KUKA KRL program: EPS_2_251524_MH1A_A_20251121061154.src

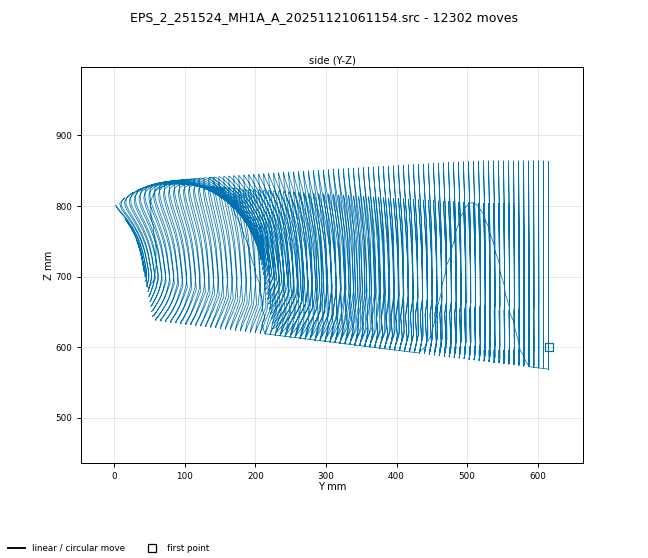
[picture p0: tool path of EPS_2_251524_MH1A_A_20251121061154.src, 12302 of 12304 moves have a stored position in this frame; points joined in program order, loops and branches not executed]
&ACCESS RVP
&REL 4
&COMMENT QRS 19112012
&PARAM EDITMASK = *
DEF PART()
EXT BAS (BAS_COMMAND :IN,REAL :IN )
INT I
BAS (#INITMOV,0 )

;KUKA QRS Post kuka4.cps  Date:22-06-2017 !

File_ID=2928

QRS_PRE_INIT()

;Init var - Until changes are made in qrs_pre_init
Outlet_Square_prg=0
Inlet_1_Square_prg=0
Inlet_2_Square_prg=0
Inlet_3_Square_prg=0
Inlet_4_Square_prg=0
Inlet_5_Square_prg=0

Outlet_1={X 0.000, Y 513.730, Z 763.500, B 0.000, E1 0.000 }
Inlet_1={X 0.000, Y 518.010, Z 703.500, B 0.000, E1 125.000 }
Outlet_1_type=201
Inlet_1_type=201
;QRS#1=Sidecore dimensions
;QRS#2=200-8" PVC SDR 35
;QRS#3=200-8" PVC SDR 35
;QRS#4=
;QRS#5=
;QRS#6=
;QRS#7=
;QRS#8=
;QRS#9=12-08 PSX
;QRS#10=12-08 PSX
;QRS#11=
;QRS#12=
;QRS#13=
;QRS#14=
;QRS#15=
;QRS#16=1220x127x1143 3,75'
;QRS#17=EPS Height
;QRS#18=864
;QRS#19=*
;QRS#20= UPDATED VERSION 22-06-2017
;QRS#21=*
Outlet_Square=0100
Inlet_1_Square=0100
Inlet_2_Square=0
Inlet_3_Square=0
Inlet_4_Square=0
Inlet_5_Square=0
Mill_Square=1
Outlet_Square_Prg=204
Inlet_1_Square_prg=204

QRS_INIT()

$ADVANCE=5

; T1
PTP {E1 173.595,E2 173.595}
PTP {X 0,Y 615.511,A -85,B 0,C 180,E1 173.595,E2 173.595,E3 0,E4 0,E5 0,E6 0}
QRS_SPEED_INIT()
LIN {X 0,Y 615.511,Z 600,A -85,B 0,C 180,E1 173.595,E2 173.595,E3 0,E4 0,E5 0,E6 0} C_VEL
LIN {X 0,Y 615.511,Z 578.873,A -85,B 0,C 180,E1 173.595,E2 173.595} C_VEL
LIN {X 0,Y 615.511,Z 570.691,A -85,B 0,C 180,E1 173.595,E2 173.595} C_VEL
LIN {X 0,Y 615.492,Z 568.691,A -85,B 0,C 180,E1 173.409,E2 173.409} C_VEL
LIN {X 0,Y 615.475,Z 568.685,A -85,B 0,C 180,E1 170.801,E2 170.801} C_VEL
LIN {X 0,Y 615.486,Z 568.69,A -85,B 0,C 180,E1 168.139,E2 168.139} C_VEL
LIN {X 0,Y 615.493,Z 568.691,A -85,B 0,C 180,E1 165.451,E2 165.451} C_VEL
LIN {X 0,Y 615.476,Z 568.685,A -85,B 0,C 180,E1 162.729,E2 162.729} C_VEL
LIN {X 0,Y 615.485,Z 568.748,A -85,B 0,C 180,E1 162.301,E2 162.301} C_VEL
LIN {X 0,Y 615.48,Z 584.538,A -85,B 0,C 180,E1 159.442,E2 159.442} C_VEL
LIN {X 0,Y 615.48,Z 593.631,A -85,B 0,C 180,E1 157.811,E2 157.811} C_VEL
LIN {X 0,Y 615.477,Z 700.494,A -85,B 0,C 180,E1 156.532,E2 156.532} C_VEL
LIN {X 0,Y 615.486,Z 713.363,A -85,B 0,C 180,E1 156.245,E2 156.245} C_VEL
LIN {X 0,Y 615.488,Z 725.164,A -85,B 0,C 180,E1 155.859,E2 155.859} C_VEL
LIN {X 0,Y 615.492,Z 736.391,A -85,B 0,C 180,E1 155.369,E2 155.369} C_VEL
LIN {X 0,Y 615.486,Z 747.967,A -85,B 0,C 180,E1 154.718,E2 154.718} C_VEL
LIN {X 0,Y 615.499,Z 759.136,A -85,B 0,C 180,E1 153.921,E2 153.921} C_VEL
LIN {X 0,Y 615.499,Z 768.418,A -85,B 0,C 180,E1 153.103,E2 153.103} C_VEL
LIN {X 0,Y 615.493,Z 777.665,A -85,B 0,C 180,E1 152.085,E2 152.085} C_VEL
LIN {X 0,Y 615.498,Z 784.494,A -85,B 0,C 180,E1 151.156,E2 151.156} C_VEL
LIN {X 0,Y 615.499,Z 790.175,A -85,B 0,C 180,E1 150.202,E2 150.202} C_VEL
LIN {X 0,Y 615.497,Z 795.401,A -85,B 0,C 180,E1 149.081,E2 149.081} C_VEL
LIN {X 0,Y 615.495,Z 798.12,A -85,B 0,C 180,E1 148.315,E2 148.315} C_VEL
LIN {X 0,Y 615.493,Z 800.307,A -85,B 0,C 180,E1 147.543,E2 147.543} C_VEL
LIN {X 0,Y 615.495,Z 802.346,A -85,B 0,C 180,E1 146.463,E2 146.463} C_VEL
LIN {X 0,Y 615.492,Z 803.34,A -85,B 0,C 180,E1 145.185,E2 145.185} C_VEL
LIN {X 0,Y 615.496,Z 803.076,A -85,B 0,C 180,E1 144.163,E2 144.163} C_VEL
LIN {X 0,Y 615.493,Z 801.724,A -85,B 0,C 180,E1 143.061,E2 143.061} C_VEL
LIN {X 0,Y 615.495,Z 799.15,A -85,B 0,C 180,E1 141.932,E2 141.932} C_VEL
LIN {X 0,Y 615.496,Z 795.8,A -85,B 0,C 180,E1 140.935,E2 140.935} C_VEL
LIN {X 0,Y 615.496,Z 791.221,A -85,B 0,C 180,E1 139.909,E2 139.909} C_VEL
LIN {X 0,Y 615.495,Z 785.487,A -85,B 0,C 180,E1 138.903,E2 138.903} C_VEL
LIN {X 0,Y 615.494,Z 778.427,A -85,B 0,C 180,E1 137.918,E2 137.918} C_VEL
LIN {X 0,Y 615.495,Z 769.828,A -85,B 0,C 180,E1 136.95,E2 136.95} C_VEL
LIN {X 0,Y 615.495,Z 760.482,A -85,B 0,C 180,E1 136.095,E2 136.095} C_VEL
LIN {X 0,Y 615.49,Z 750.585,A -85,B 0,C 180,E1 135.363,E2 135.363} C_VEL
LIN {X 0,Y 615.489,Z 740.106,A -85,B 0,C 180,E1 134.734,E2 134.734} C_VEL
LIN {X 0,Y 615.49,Z 727.652,A -85,B 0,C 180,E1 134.148,E2 134.148} C_VEL
LIN {X 0,Y 615.496,Z 715.095,A -85,B 0,C 180,E1 133.713,E2 133.713} C_VEL
LIN {X 0,Y 615.479,Z 702.164,A -85,B 0,C 180,E1 133.408,E2 133.408} C_VEL
LIN {X 0,Y 615.477,Z 680.151,A -85,B 0,C 180,E1 133.121,E2 133.121} C_VEL
LIN {X 0,Y 615.477,Z 593.615,A -85,B 0,C 180,E1 132.096,E2 132.096} C_VEL
LIN {X 0,Y 615.482,Z 578.635,A -85,B 0,C 180,E1 129.404,E2 129.404} C_VEL
LIN {X 0,Y 615.49,Z 568.685,A -85,B 0,C 180,E1 127.577,E2 127.577} C_VEL
LIN {X 0,Y 615.49,Z 568.684,A -85,B 0,C 180,E1 124.701,E2 124.701} C_VEL
LIN {X 0,Y 615.492,Z 568.691,A -85,B 0,C 180,E1 122.331,E2 122.331} C_VEL
LIN {X 0,Y 615.492,Z 568.684,A -85,B 0,C 180,E1 119.405,E2 119.405} C_VEL
LIN {X 0,Y 615.474,Z 568.684,A -85,B 0,C 180,E1 117.043,E2 117.043} C_VEL
LIN {X 0,Y 615.495,Z 568.688,A -85,B 0,C 180,E1 114.271,E2 114.271} C_VEL
LIN {X 0,Y 615.492,Z 568.688,A -85,B 0,C 180,E1 111.431,E2 111.431} C_VEL
LIN {X 0,Y 615.478,Z 568.684,A -85,B 0,C 180,E1 108.602,E2 108.602} C_VEL
LIN {X 0,Y 615.492,Z 568.696,A -85,B 0,C 180,E1 105.904,E2 105.904} C_VEL
LIN {X 0,Y 615.497,Z 568.684,A -85,B 0,C 180,E1 103.2,E2 103.2} C_VEL
LIN {X 0,Y 615.476,Z 568.684,A -85,B 0,C 180,E1 100.526,E2 100.526} C_VEL
LIN {X 0,Y 615.493,Z 568.691,A -85,B 0,C 180,E1 97.875,E2 97.875} C_VEL
LIN {X 0,Y 615.486,Z 568.692,A -85,B 0,C 180,E1 95.24,E2 95.24} C_VEL
LIN {X 0,Y 615.477,Z 568.684,A -85,B 0,C 180,E1 92.617,E2 92.617} C_VEL
LIN {X 0,Y 615.489,Z 568.685,A -85,B 0,C 180,E1 89.999,E2 89.999} C_VEL
LIN {X 0,Y 615.495,Z 568.7,A -85,B 0,C 180,E1 87.381,E2 87.381} C_VEL
LIN {X 0,Y 615.485,Z 568.685,A -85,B 0,C 180,E1 84.758,E2 84.758} C_VEL
LIN {X 0,Y 615.481,Z 568.683,A -85,B 0,C 180,E1 82.124,E2 82.124} C_VEL
LIN {X 0,Y 615.49,Z 568.694,A -85,B 0,C 180,E1 79.472,E2 79.472} C_VEL
LIN {X 0,Y 615.497,Z 568.686,A -85,B 0,C 180,E1 76.798,E2 76.798} C_VEL
LIN {X 0,Y 615.478,Z 568.683,A -85,B 0,C 180,E1 74.094,E2 74.094} C_VEL
LIN {X 0,Y 615.491,Z 568.693,A -85,B 0,C 180,E1 71.353,E2 71.353} C_VEL
LIN {X 0,Y 615.492,Z 568.686,A -85,B 0,C 180,E1 68.568,E2 68.568} C_VEL
LIN {X 0,Y 615.489,Z 568.682,A -85,B 0,C 180,E1 65.727,E2 65.727} C_VEL
LIN {X 0,Y 615.494,Z 568.696,A -85,B 0,C 180,E1 62.823,E2 62.823} C_VEL
LIN {X 0,Y 615.476,Z 568.685,A -85,B 0,C 180,E1 60.207,E2 60.207} C_VEL
LIN {X 0,Y 615.486,Z 568.684,A -85,B 0,C 180,E1 57.542,E2 57.542} C_VEL
LIN {X 0,Y 615.492,Z 568.689,A -85,B 0,C 180,E1 55.185,E2 55.185} C_VEL
LIN {X 0,Y 615.491,Z 568.701,A -85,B 0,C 180,E1 52.758,E2 52.758} C_VEL
LIN {X 0,Y 615.477,Z 568.684,A -85,B 0,C 180,E1 49.912,E2 49.912} C_VEL
LIN {X 0,Y 615.478,Z 568.683,A -85,B 0,C 180,E1 47.646,E2 47.646} C_VEL
LIN {X 0,Y 615.49,Z 568.691,A -85,B 0,C 180,E1 44.931,E2 44.931} C_VEL
LIN {X 0,Y 615.49,Z 568.686,A -85,B 0,C 180,E1 42.08,E2 42.08} C_VEL
LIN {X 0,Y 615.474,Z 568.685,A -85,B 0,C 180,E1 39.751,E2 39.751} C_VEL
LIN {X 0,Y 615.489,Z 568.687,A -85,B 0,C 180,E1 36.936,E2 36.936} C_VEL
LIN {X 0,Y 615.495,Z 568.687,A -85,B 0,C 180,E1 34.021,E2 34.021} C_VEL
LIN {X 0,Y 615.478,Z 568.685,A -85,B 0,C 180,E1 31.686,E2 31.686} C_VEL
LIN {X 0,Y 615.477,Z 568.683,A -85,B 0,C 180,E1 29.407,E2 29.407} C_VEL
LIN {X 0,Y 615.488,Z 568.682,A -85,B 0,C 180,E1 27.044,E2 27.044} C_VEL
LIN {X 0,Y 615.488,Z 568.702,A -85,B 0,C 180,E1 24.272,E2 24.272} C_VEL
LIN {X 0,Y 615.477,Z 568.685,A -85,B 0,C 180,E1 21.432,E2 21.432} C_VEL
LIN {X 0,Y 615.486,Z 568.687,A -85,B 0,C 180,E1 18.646,E2 18.646} C_VEL
LIN {X 0,Y 615.489,Z 568.695,A -85,B 0,C 180,E1 15.905,E2 15.905} C_VEL
LIN {X 0,Y 615.476,Z 568.684,A -85,B 0,C 180,E1 13.201,E2 13.201} C_VEL
LIN {X 0,Y 615.489,Z 568.685,A -85,B 0,C 180,E1 10.527,E2 10.527} C_VEL
LIN {X 0,Y 615.493,Z 568.698,A -85,B 0,C 180,E1 7.875,E2 7.875} C_VEL
LIN {X 0,Y 615.478,Z 568.686,A -85,B 0,C 180,E1 5.241,E2 5.241} C_VEL
LIN {X 0,Y 615.494,Z 568.681,A -85,B 0,C 180,E1 2.618,E2 2.618} C_VEL
LIN {X 0,Y 615.491,Z 568.695,A -85,B 0,C 180,E1 0,E2 0} C_VEL
LIN {X 0,Y 615.494,Z 568.688,A -85,B 0,C 180,E1 -2.618,E2 -2.618} C_VEL
LIN {X 0,Y 615.477,Z 568.683,A -85,B 0,C 180,E1 -5.241,E2 -5.241} C_VEL
LIN {X 0,Y 615.489,Z 568.687,A -85,B 0,C 180,E1 -7.876,E2 -7.876} C_VEL
LIN {X 0,Y 615.484,Z 568.687,A -85,B 0,C 180,E1 -10.885,E2 -10.885} C_VEL
LIN {X 0,Y 615.476,Z 568.685,A -85,B 0,C 180,E1 -13.202,E2 -13.202} C_VEL
LIN {X 0,Y 615.487,Z 568.685,A -85,B 0,C 180,E1 -15.905,E2 -15.905} C_VEL
LIN {X 0,Y 615.494,Z 568.697,A -85,B 0,C 180,E1 -18.646,E2 -18.646} C_VEL
LIN {X 0,Y 615.476,Z 568.684,A -85,B 0,C 180,E1 -21.432,E2 -21.432} C_VEL
LIN {X 0,Y 615.487,Z 568.69,A -85,B 0,C 180,E1 -24.272,E2 -24.272} C_VEL
LIN {X 0,Y 615.48,Z 568.688,A -85,B 0,C 180,E1 -27.178,E2 -27.178} C_VEL
LIN {X 0,Y 615.485,Z 568.682,A -85,B 0,C 180,E1 -29.793,E2 -29.793} C_VEL
LIN {X 0,Y 615.487,Z 568.691,A -85,B 0,C 180,E1 -32.458,E2 -32.458} C_VEL
LIN {X 0,Y 615.498,Z 568.7,A -85,B 0,C 180,E1 -34.815,E2 -34.815} C_VEL
LIN {X 0,Y 615.49,Z 568.689,A -85,B 0,C 180,E1 -37.242,E2 -37.242} C_VEL
LIN {X 0,Y 615.493,Z 568.68,A -85,B 0,C 180,E1 -40.089,E2 -40.089} C_VEL
LIN {X 0,Y 615.496,Z 568.698,A -85,B 0,C 180,E1 -43.048,E2 -43.048} C_VEL
LIN {X 0,Y 615.481,Z 568.682,A -85,B 0,C 180,E1 -46.003,E2 -46.003} C_VEL
LIN {X 0,Y 615.489,Z 568.696,A -85,B 0,C 180,E1 -48.906,E2 -48.906} C_VEL
LIN {X 0,Y 615.495,Z 568.7,A -85,B 0,C 180,E1 -51.096,E2 -51.096} C_VEL
LIN {X 0,Y 615.482,Z 568.69,A -85,B 0,C 180,E1 -53.574,E2 -53.574} C_VEL
LIN {X 0,Y 615.475,Z 568.685,A -85,B 0,C 180,E1 -55.977,E2 -55.977} C_VEL
LIN {X 0,Y 615.487,Z 568.681,A -85,B 0,C 180,E1 -58.314,E2 -58.314} C_VEL
LIN {X 0,Y 615.494,Z 568.681,A -85,B 0,C 180,E1 -60.593,E2 -60.593} C_VEL
LIN {X 0,Y 615.494,Z 568.693,A -85,B 0,C 180,E1 -63.556,E2 -63.556} C_VEL
LIN {X 0,Y 615.487,Z 568.681,A -85,B 0,C 180,E1 -66.443,E2 -66.443} C_VEL
LIN {X 0,Y 615.492,Z 568.868,A -85,B 0,C 180,E1 -66.711,E2 -66.711} C_VEL
LIN {X 0,Y 615.487,Z 591.047,A -85,B 0,C 180,E1 -69.575,E2 -69.575} C_VEL
LIN {X 0,Y 615.484,Z 613.193,A -85,B 0,C 180,E1 -72.386,E2 -72.386} C_VEL
LIN {X 0,Y 615.481,Z 634.978,A -85,B 0,C 180,E1 -75.112,E2 -75.112} C_VEL
LIN {X 0,Y 615.478,Z 651.127,A -85,B 0,C 180,E1 -77.113,E2 -77.113} C_VEL
LIN {X 0,Y 615.476,Z 759.796,A -85,B 0,C 180,E1 -78.41,E2 -78.41} C_VEL
LIN {X 0,Y 615.487,Z 772.32,A -85,B 0,C 180,E1 -78.681,E2 -78.681} C_VEL
LIN {X 0,Y 615.496,Z 785.511,A -85,B 0,C 180,E1 -79.109,E2 -79.109} C_VEL
LIN {X 0,Y 615.484,Z 797.465,A -85,B 0,C 180,E1 -79.639,E2 -79.639} C_VEL
LIN {X 0,Y 615.483,Z 808.986,A -85,B 0,C 180,E1 -80.303,E2 -80.303} C_VEL
LIN {X 0,Y 615.499,Z 819.333,A -85,B 0,C 180,E1 -81.049,E2 -81.049} C_VEL
LIN {X 0,Y 615.497,Z 827.805,A -85,B 0,C 180,E1 -81.793,E2 -81.793} C_VEL
LIN {X 0,Y 615.498,Z 835.6,A -85,B 0,C 180,E1 -82.619,E2 -82.619} C_VEL
LIN {X 0,Y 615.496,Z 843.198,A -85,B 0,C 180,E1 -83.607,E2 -83.607} C_VEL
LIN {X 0,Y 615.498,Z 850.201,A -85,B 0,C 180,E1 -84.758,E2 -84.758} C_VEL
LIN {X 0,Y 615.494,Z 854.848,A -85,B 0,C 180,E1 -85.743,E2 -85.743} C_VEL
LIN {X 0,Y 615.496,Z 858.396,A -85,B 0,C 180,E1 -86.726,E2 -86.726} C_VEL
LIN {X 0,Y 615.497,Z 860.231,A -85,B 0,C 180,E1 -87.381,E2 -87.381} C_VEL
LIN {X 0,Y 615.496,Z 861.607,A -85,B 0,C 180,E1 -88.036,E2 -88.036} C_VEL
LIN {X 0,Y 615.496,Z 863.173,A -85,B 0,C 180,E1 -89.345,E2 -89.345} C_VEL
LIN {X 0,Y 615.494,Z 863.389,A -85,B 0,C 180,E1 -89.999,E2 -89.999} C_VEL
LIN {X 0,Y 615.496,Z 862.581,A -85,B 0,C 180,E1 -91.308,E2 -91.308} C_VEL
LIN {X 0,Y 615.496,Z 861.609,A -85,B 0,C 180,E1 -91.962,E2 -91.962} C_VEL
LIN {X 0,Y 615.497,Z 860.235,A -85,B 0,C 180,E1 -92.617,E2 -92.617} C_VEL
LIN {X 0,Y 615.496,Z 857.352,A -85,B 0,C 180,E1 -93.6,E2 -93.6} C_VEL
LIN {X 0,Y 615.498,Z 853.445,A -85,B 0,C 180,E1 -94.584,E2 -94.584} C_VEL
LIN {X 0,Y 615.499,Z 848.409,A -85,B 0,C 180,E1 -95.569,E2 -95.569} C_VEL
LIN {X 0,Y 615.497,Z 841.87,A -85,B 0,C 180,E1 -96.583,E2 -96.583} C_VEL
LIN {X 0,Y 615.497,Z 834.14,A -85,B 0,C 180,E1 -97.545,E2 -97.545} C_VEL
LIN {X 0,Y 615.498,Z 826.053,A -85,B 0,C 180,E1 -98.37,E2 -98.37} C_VEL
LIN {X 0,Y 615.499,Z 816.178,A -85,B 0,C 180,E1 -99.198,E2 -99.198} C_VEL
LIN {X 0,Y 615.487,Z 804.995,A -85,B 0,C 180,E1 -99.944,E2 -99.944} C_VEL
LIN {X 0,Y 615.483,Z 794.039,A -85,B 0,C 180,E1 -100.526,E2 -100.526} C_VEL
LIN {X 0,Y 615.496,Z 781.443,A -85,B 0,C 180,E1 -101.041,E2 -101.041} C_VEL
LIN {X 0,Y 615.482,Z 769.101,A -85,B 0,C 180,E1 -101.401,E2 -101.401} C_VEL
LIN {X 0,Y 615.475,Z 755.527,A -85,B 0,C 180,E1 -101.651,E2 -101.651} C_VEL
LIN {X 0,Y 615.478,Z 651.139,A -85,B 0,C 180,E1 -102.886,E2 -102.886} C_VEL
LIN {X 0,Y 615.48,Z 629.545,A -85,B 0,C 180,E1 -105.565,E2 -105.565} C_VEL
LIN {X 0,Y 615.498,Z 607.928,A -85,B 0,C 180,E1 -108.278,E2 -108.278} C_VEL
LIN {X 0,Y 615.495,Z 585.938,A -85,B 0,C 180,E1 -111.08,E2 -111.08} C_VEL
LIN {X 0,Y 615.496,Z 568.681,A -85,B 0,C 180,E1 -113.332,E2 -113.332} C_VEL
LIN {X 0,Y 615.48,Z 568.684,A -85,B 0,C 180,E1 -115.715,E2 -115.715} C_VEL
LIN {X 0,Y 615.495,Z 568.697,A -85,B 0,C 180,E1 -118.451,E2 -118.451} C_VEL
LIN {X 0,Y 615.475,Z 568.689,A -85,B 0,C 180,E1 -121.084,E2 -121.084} C_VEL
LIN {X 0,Y 615.495,Z 568.68,A -85,B 0,C 180,E1 -123.535,E2 -123.535} C_VEL
LIN {X 0,Y 615.483,Z 568.7,A -85,B 0,C 180,E1 -126.424,E2 -126.424} C_VEL
LIN {X 0,Y 615.476,Z 568.689,A -85,B 0,C 180,E1 -129.06,E2 -129.06} C_VEL
LIN {X 0,Y 615.481,Z 568.683,A -85,B 0,C 180,E1 -131.473,E2 -131.473} C_VEL
LIN {X 0,Y 615.482,Z 568.692,A -85,B 0,C 180,E1 -134.149,E2 -134.149} C_VEL
LIN {X 0,Y 615.484,Z 568.689,A -85,B 0,C 180,E1 -136.952,E2 -136.952} C_VEL
LIN {X 0,Y 615.473,Z 568.685,A -85,B 0,C 180,E1 -139.392,E2 -139.392} C_VEL
LIN {X 0,Y 615.49,Z 568.687,A -85,B 0,C 180,E1 -141.986,E2 -141.986} C_VEL
LIN {X 0,Y 615.495,Z 568.698,A -85,B 0,C 180,E1 -144.384,E2 -144.384} C_VEL
LIN {X 0,Y 615.482,Z 568.693,A -85,B 0,C 180,E1 -146.763,E2 -146.763} C_VEL
LIN {X 0,Y 615.485,Z 568.685,A -85,B 0,C 180,E1 -149.08,E2 -149.08} C_VEL
LIN {X 0,Y 615.476,Z 568.685,A -85,B 0,C 180,E1 -151.55,E2 -151.55} C_VEL
LIN {X 0,Y 615.496,Z 568.7,A -85,B 0,C 180,E1 -154.427,E2 -154.427} C_VEL
LIN {X 0,Y 615.486,Z 568.684,A -85,B 0,C 180,E1 -157.155,E2 -157.155} C_VEL
LIN {X 0,Y 615.485,Z 568.69,A -85,B 0,C 180,E1 -159.967,E2 -159.967} C_VEL
LIN {X 0,Y 615.476,Z 568.693,A -85,B 0,C 180,E1 -162.729,E2 -162.729} C_VEL
LIN {X 0,Y 615.48,Z 568.684,A -85,B 0,C 180,E1 -165.451,E2 -165.451} C_VEL
LIN {X 0,Y 615.486,Z 568.695,A -85,B 0,C 180,E1 -168.139,E2 -168.139} C_VEL
LIN {X 0,Y 615.475,Z 568.691,A -85,B 0,C 180,E1 -170.801,E2 -170.801} C_VEL
LIN {X 0,Y 615.488,Z 568.682,A -85,B 0,C 180,E1 -173.443,E2 -173.443} C_VEL
LIN {X 0,Y 615.478,Z 568.696,A -85,B 0,C 180,E1 -176.071,E2 -176.071} C_VEL
LIN {X 0,Y 615.484,Z 568.691,A -85,B 0,C 180,E1 -178.691,E2 -178.691} C_VEL
LIN {X 0,Y 615.484,Z 568.683,A -85,B 0,C 180,E1 -181.309,E2 -181.309} C_VEL
LIN {X 0,Y 615.478,Z 568.693,A -85,B 0,C 180,E1 -183.928,E2 -183.928} C_VEL
LIN {X 0,Y 615.492,Z 568.691,A -85,B 0,C 180,E1 -186.591,E2 -186.591} C_VEL
LIN {X 0,Y 614.805,Z 568.832,A -85,B 0,C 180,E1 -187.137,E2 -187.137} C_VEL
LIN {X 0,Y 611.961,Z 569.256,A -85,B 0,C 180,E1 -188.023,E2 -188.023} C_VEL
LIN {X 0,Y 609.569,Z 569.562,A -85,B 0,C 180,E1 -188.735,E2 -188.735} C_VEL
LIN {X 0,Y 608.539,Z 569.678,A -85,B 0,C 180,E1 -189.285,E2 -189.285} C_VEL
LIN {X 0,Y 608.452,Z 569.688,A -85,B 0,C 180,E1 -189.471,E2 -189.471} C_VEL
LIN {X 0,Y 608.462,Z 569.692,A -85,B 0,C 180,E1 -192,E2 -192} C_VEL
LIN {X 0,Y 608.476,Z 569.688,A -85,B 0,C 180,E1 -194.72,E2 -194.72} C_VEL
LIN {X 0,Y 608.46,Z 569.708,A -85,B 0,C 180,E1 -197.65,E2 -197.65} C_VEL
LIN {X 0,Y 608.459,Z 584.081,A -85,B 0,C 180,E1 -200.274,E2 -200.274} C_VEL
LIN {X 0,Y 608.445,Z 593.907,A -85,B 0,C 180,E1 -202.049,E2 -202.049} C_VEL
LIN {X 0,Y 608.541,Z 700.018,A -85,B 0,C 180,E1 -203.323,E2 -203.323} C_VEL
LIN {X 0,Y 608.541,Z 713.172,A -85,B 0,C 180,E1 -203.616,E2 -203.616} C_VEL
LIN {X 0,Y 608.527,Z 725.294,A -85,B 0,C 180,E1 -204.015,E2 -204.015} C_VEL
LIN {X 0,Y 608.522,Z 737.703,A -85,B 0,C 180,E1 -204.568,E2 -204.568} C_VEL
LIN {X 0,Y 608.474,Z 748.78,A -85,B 0,C 180,E1 -205.208,E2 -205.208} C_VEL
LIN {X 0,Y 608.473,Z 760.146,A -85,B 0,C 180,E1 -206.034,E2 -206.034} C_VEL
LIN {X 0,Y 608.465,Z 769.943,A -85,B 0,C 180,E1 -206.927,E2 -206.927} C_VEL
LIN {X 0,Y 608.463,Z 778.517,A -85,B 0,C 180,E1 -207.891,E2 -207.891} C_VEL
LIN {X 0,Y 608.46,Z 785.022,A -85,B 0,C 180,E1 -208.787,E2 -208.787} C_VEL
LIN {X 0,Y 608.448,Z 790.886,A -85,B 0,C 180,E1 -209.781,E2 -209.781} C_VEL
LIN {X 0,Y 608.429,Z 796.071,A -85,B 0,C 180,E1 -210.908,E2 -210.908} C_VEL
LIN {X 0,Y 608.419,Z 800.011,A -85,B 0,C 180,E1 -212.097,E2 -212.097} C_VEL
LIN {X 0,Y 608.433,Z 801.87,A -85,B 0,C 180,E1 -212.881,E2 -212.881} C_VEL
LIN {X 0,Y 608.419,Z 803.193,A -85,B 0,C 180,E1 -213.729,E2 -213.729} C_VEL
LIN {X 0,Y 608.417,Z 803.973,A -85,B 0,C 180,E1 -214.903,E2 -214.903} C_VEL
LIN {X 0,Y 608.447,Z 803.505,A -85,B 0,C 180,E1 -216.092,E2 -216.092} C_VEL
LIN {X 0,Y 608.434,Z 801.983,A -85,B 0,C 180,E1 -217.156,E2 -217.156} C_VEL
LIN {X 0,Y 608.425,Z 799.336,A -85,B 0,C 180,E1 -218.237,E2 -218.237} C_VEL
LIN {X 0,Y 608.452,Z 794.985,A -85,B 0,C 180,E1 -219.441,E2 -219.441} C_VEL
LIN {X 0,Y 608.443,Z 789.732,A -85,B 0,C 180,E1 -220.521,E2 -220.521} C_VEL
LIN {X 0,Y 608.452,Z 783.819,A -85,B 0,C 180,E1 -221.482,E2 -221.482} C_VEL
LIN {X 0,Y 608.473,Z 776.484,A -85,B 0,C 180,E1 -222.448,E2 -222.448} C_VEL
LIN {X 0,Y 608.475,Z 767.471,A -85,B 0,C 180,E1 -223.407,E2 -223.407} C_VEL
LIN {X 0,Y 608.477,Z 757.47,A -85,B 0,C 180,E1 -224.267,E2 -224.267} C_VEL
LIN {X 0,Y 608.481,Z 746.954,A -85,B 0,C 180,E1 -224.999,E2 -224.999} C_VEL
LIN {X 0,Y 608.504,Z 735.104,A -85,B 0,C 180,E1 -225.649,E2 -225.649} C_VEL
LIN {X 0,Y 608.527,Z 722.609,A -85,B 0,C 180,E1 -226.176,E2 -226.176} C_VEL
LIN {X 0,Y 608.537,Z 709.783,A -85,B 0,C 180,E1 -226.565,E2 -226.565} C_VEL
LIN {X 0,Y 608.543,Z 697.399,A -85,B 0,C 180,E1 -226.807,E2 -226.807} C_VEL
LIN {X 0,Y 608.47,Z 594.096,A -85,B 0,C 180,E1 -228.038,E2 -228.038} C_VEL
LIN {X 0,Y 608.473,Z 579.203,A -85,B 0,C 180,E1 -230.702,E2 -230.702} C_VEL
LIN {X 0,Y 608.478,Z 569.686,A -85,B 0,C 180,E1 -232.459,E2 -232.459} C_VEL
LIN {X 0,Y 608.475,Z 569.684,A -85,B 0,C 180,E1 -235.091,E2 -235.091} C_VEL
LIN {X 0,Y 608.471,Z 569.695,A -85,B 0,C 180,E1 -237.907,E2 -237.907} C_VEL
LIN {X 0,Y 608.465,Z 569.692,A -85,B 0,C 180,E1 -240.221,E2 -240.221} C_VEL
LIN {X 0,Y 608.472,Z 569.685,A -85,B 0,C 180,E1 -242.794,E2 -242.794} C_VEL
LIN {X 0,Y 608.453,Z 569.688,A -85,B 0,C 180,E1 -245.43,E2 -245.43} C_VEL
LIN {X 0,Y 608.474,Z 569.692,A -85,B 0,C 180,E1 -248.31,E2 -248.31} C_VEL
LIN {X 0,Y 608.452,Z 569.687,A -85,B 0,C 180,E1 -251.131,E2 -251.131} C_VEL
LIN {X 0,Y 608.464,Z 569.69,A -85,B 0,C 180,E1 -253.907,E2 -253.907} C_VEL
LIN {X 0,Y 608.473,Z 569.689,A -85,B 0,C 180,E1 -256.645,E2 -256.645} C_VEL
LIN {X 0,Y 608.456,Z 569.686,A -85,B 0,C 180,E1 -259.351,E2 -259.351} C_VEL
LIN {X 0,Y 608.482,Z 569.688,A -85,B 0,C 180,E1 -262.034,E2 -262.034} C_VEL
LIN {X 0,Y 608.466,Z 569.692,A -85,B 0,C 180,E1 -264.699,E2 -264.699} C_VEL
LIN {X 0,Y 608.469,Z 569.685,A -85,B 0,C 180,E1 -267.353,E2 -267.353} C_VEL
LIN {X 0,Y 608.48,Z 569.686,A -85,B 0,C 180,E1 -270.001,E2 -270.001} C_VEL
LIN {X 0,Y 608.485,Z 569.693,A -85,B 0,C 180,E1 -272.649,E2 -272.649} C_VEL
LIN {X 0,Y 608.464,Z 569.686,A -85,B 0,C 180,E1 -275.303,E2 -275.303} C_VEL
LIN {X 0,Y 608.476,Z 569.685,A -85,B 0,C 180,E1 -277.968,E2 -277.968} C_VEL
LIN {X 0,Y 608.469,Z 569.694,A -85,B 0,C 180,E1 -280.65,E2 -280.65} C_VEL
LIN {X 0,Y 608.47,Z 569.687,A -85,B 0,C 180,E1 -283.357,E2 -283.357} C_VEL
LIN {X 0,Y 608.459,Z 569.687,A -85,B 0,C 180,E1 -286.095,E2 -286.095} C_VEL
LIN {X 0,Y 608.459,Z 569.697,A -85,B 0,C 180,E1 -288.87,E2 -288.87} C_VEL
LIN {X 0,Y 608.469,Z 569.685,A -85,B 0,C 180,E1 -291.692,E2 -291.692} C_VEL
LIN {X 0,Y 608.458,Z 569.69,A -85,B 0,C 180,E1 -294.571,E2 -294.571} C_VEL
LIN {X 0,Y 608.487,Z 569.691,A -85,B 0,C 180,E1 -297.209,E2 -297.209} C_VEL
LIN {X 0,Y 608.459,Z 569.686,A -85,B 0,C 180,E1 -299.97,E2 -299.97} C_VEL
LIN {X 0,Y 608.457,Z 569.692,A -85,B 0,C 180,E1 -302.88,E2 -302.88} C_VEL
LIN {X 0,Y 608.452,Z 569.697,A -85,B 0,C 180,E1 -305.278,E2 -305.278} C_VEL
LIN {X 0,Y 608.466,Z 569.688,A -85,B 0,C 180,E1 -307.747,E2 -307.747} C_VEL
LIN {X 0,Y 608.447,Z 569.687,A -85,B 0,C 180,E1 -310.328,E2 -310.328} C_VEL
LIN {X 0,Y 608.481,Z 569.694,A -85,B 0,C 180,E1 -313.31,E2 -313.31} C_VEL
LIN {X 0,Y 608.47,Z 569.685,A -85,B 0,C 180,E1 -316.131,E2 -316.131} C_VEL
LIN {X 0,Y 608.457,Z 569.688,A -85,B 0,C 180,E1 -318.824,E2 -318.824} C_VEL
LIN {X 0,Y 608.473,Z 569.69,A -85,B 0,C 180,E1 -321.76,E2 -321.76} C_VEL
LIN {X 0,Y 608.449,Z 569.691,A -85,B 0,C 180,E1 -323.955,E2 -323.955} C_VEL
LIN {X 0,Y 608.449,Z 569.688,A -85,B 0,C 180,E1 -326.328,E2 -326.328} C_VEL
LIN {X 0,Y 608.449,Z 569.687,A -85,B 0,C 180,E1 -328.733,E2 -328.733} C_VEL
LIN {X 0,Y 608.479,Z 569.689,A -85,B 0,C 180,E1 -331.38,E2 -331.38} C_VEL
LIN {X 0,Y 608.469,Z 569.687,A -85,B 0,C 180,E1 -334.281,E2 -334.281} C_VEL
LIN {X 0,Y 608.45,Z 569.687,A -85,B 0,C 180,E1 -336.876,E2 -336.876} C_VEL
LIN {X 0,Y 608.469,Z 569.694,A -85,B 0,C 180,E1 -339.726,E2 -339.726} C_VEL
LIN {X 0,Y 608.448,Z 569.689,A -85,B 0,C 180,E1 -342.523,E2 -342.523} C_VEL
LIN {X 0,Y 608.475,Z 569.685,A -85,B 0,C 180,E1 -345.28,E2 -345.28} C_VEL
LIN {X 0,Y 608.47,Z 569.696,A -85,B 0,C 180,E1 -348,E2 -348} C_VEL
LIN {X 0,Y 608.461,Z 569.687,A -85,B 0,C 180,E1 -350.694,E2 -350.694} C_VEL
LIN {X 0,Y 608.484,Z 569.684,A -85,B 0,C 180,E1 -353.368,E2 -353.368} C_VEL
LIN {X 0,Y 608.454,Z 569.696,A -85,B 0,C 180,E1 -356.026,E2 -356.026} C_VEL
LIN {X 0,Y 608.469,Z 569.687,A -85,B 0,C 180,E1 -358.676,E2 -358.676} C_VEL
LIN {X 0,Y 608.469,Z 569.685,A -85,B 0,C 180,E1 -361.324,E2 -361.324} C_VEL
LIN {X 0,Y 608.458,Z 569.692,A -85,B 0,C 180,E1 -363.974,E2 -363.974} C_VEL
LIN {X 0,Y 608.466,Z 569.69,A -85,B 0,C 180,E1 -366.633,E2 -366.633} C_VEL
LIN {X 0,Y 608.462,Z 569.685,A -85,B 0,C 180,E1 -369.306,E2 -369.306} C_VEL
LIN {X 0,Y 608.466,Z 569.689,A -85,B 0,C 180,E1 -372,E2 -372} C_VEL
LIN {X 0,Y 608.48,Z 569.69,A -85,B 0,C 180,E1 -374.721,E2 -374.721} C_VEL
LIN {X 0,Y 608.449,Z 569.687,A -85,B 0,C 180,E1 -377.477,E2 -377.477} C_VEL
LIN {X 0,Y 608.448,Z 569.687,A -85,B 0,C 180,E1 -379.571,E2 -379.571} C_VEL
LIN {X 0,Y 608.482,Z 569.691,A -85,B 0,C 180,E1 -382.405,E2 -382.405} C_VEL
LIN {X 0,Y 608.456,Z 569.696,A -85,B 0,C 180,E1 -384.571,E2 -384.571} C_VEL
LIN {X 0,Y 608.477,Z 569.686,A -85,B 0,C 180,E1 -387.206,E2 -387.206} C_VEL
LIN {X 0,Y 608.469,Z 569.685,A -85,B 0,C 180,E1 -389.971,E2 -389.971} C_VEL
LIN {X 0,Y 608.457,Z 569.696,A -85,B 0,C 180,E1 -392.88,E2 -392.88} C_VEL
LIN {X 0,Y 608.442,Z 569.691,A -85,B 0,C 180,E1 -395.278,E2 -395.278} C_VEL
LIN {X 0,Y 608.472,Z 569.684,A -85,B 0,C 180,E1 -397.746,E2 -397.746} C_VEL
LIN {X 0,Y 608.454,Z 569.688,A -85,B 0,C 180,E1 -400.329,E2 -400.329} C_VEL
LIN {X 0,Y 608.485,Z 569.688,A -85,B 0,C 180,E1 -403.31,E2 -403.31} C_VEL
LIN {X 0,Y 608.468,Z 569.685,A -85,B 0,C 180,E1 -406.13,E2 -406.13} C_VEL
LIN {X 0,Y 608.458,Z 569.692,A -85,B 0,C 180,E1 -408.823,E2 -408.823} C_VEL
LIN {X 0,Y 608.444,Z 569.694,A -85,B 0,C 180,E1 -411.409,E2 -411.409} C_VEL
LIN {X 0,Y 608.45,Z 569.688,A -85,B 0,C 180,E1 -413.955,E2 -413.955} C_VEL
LIN {X 0,Y 608.471,Z 569.684,A -85,B 0,C 180,E1 -416.329,E2 -416.329} C_VEL
LIN {X 0,Y 608.451,Z 569.689,A -85,B 0,C 180,E1 -418.732,E2 -418.732} C_VEL
LIN {X 0,Y 608.481,Z 569.694,A -85,B 0,C 180,E1 -421.379,E2 -421.379} C_VEL
LIN {X 0,Y 608.444,Z 569.69,A -85,B 0,C 180,E1 -423.964,E2 -423.964} C_VEL
LIN {X 0,Y 608.495,Z 569.721,A -85,B 0,C 180,E1 -426.539,E2 -426.539} C_VEL
LIN {X 0,Y 608.573,Z 585.927,A -85,B 0,C 180,E1 -428.667,E2 -428.667} C_VEL
LIN {X 0,Y 608.548,Z 607.943,A -85,B 0,C 180,E1 -431.505,E2 -431.505} C_VEL
LIN {X 0,Y 608.485,Z 629.599,A -85,B 0,C 180,E1 -434.25,E2 -434.25} C_VEL
LIN {X 0,Y 608.494,Z 651.094,A -85,B 0,C 180,E1 -436.941,E2 -436.941} C_VEL
LIN {X 0,Y 608.551,Z 652.087,A -85,B 0,C 180,E1 -436.985,E2 -436.985} C_VEL
LIN {X 0,Y 608.532,Z 759.911,A -85,B 0,C 180,E1 -438.276,E2 -438.276} C_VEL
LIN {X 0,Y 608.536,Z 773.192,A -85,B 0,C 180,E1 -438.571,E2 -438.571} C_VEL
LIN {X 0,Y 608.544,Z 786.333,A -85,B 0,C 180,E1 -439.009,E2 -439.009} C_VEL
LIN {X 0,Y 608.501,Z 797.622,A -85,B 0,C 180,E1 -439.518,E2 -439.518} C_VEL
LIN {X 0,Y 608.474,Z 809.187,A -85,B 0,C 180,E1 -440.19,E2 -440.19} C_VEL
LIN {X 0,Y 608.485,Z 819.585,A -85,B 0,C 180,E1 -440.945,E2 -440.945} C_VEL
LIN {X 0,Y 608.475,Z 828.105,A -85,B 0,C 180,E1 -441.698,E2 -441.698} C_VEL
LIN {X 0,Y 608.471,Z 835.954,A -85,B 0,C 180,E1 -442.533,E2 -442.533} C_VEL
LIN {X 0,Y 608.461,Z 843.284,A -85,B 0,C 180,E1 -443.484,E2 -443.484} C_VEL
LIN {X 0,Y 608.45,Z 848.862,A -85,B 0,C 180,E1 -444.365,E2 -444.365} C_VEL
LIN {X 0,Y 608.432,Z 853.947,A -85,B 0,C 180,E1 -445.361,E2 -445.361} C_VEL
LIN {X 0,Y 608.449,Z 857.894,A -85,B 0,C 180,E1 -446.357,E2 -446.357} C_VEL
LIN {X 0,Y 608.425,Z 860.807,A -85,B 0,C 180,E1 -447.351,E2 -447.351} C_VEL
LIN {X 0,Y 608.441,Z 862.2,A -85,B 0,C 180,E1 -448.013,E2 -448.013} C_VEL
LIN {X 0,Y 608.439,Z 863.783,A -85,B 0,C 180,E1 -449.337,E2 -449.337} C_VEL
LIN {X 0,Y 608.434,Z 864,A -85,B 0,C 180,E1 -449.999,E2 -449.999} C_VEL
LIN {X 0,Y 608.448,Z 863.185,A -85,B 0,C 180,E1 -451.323,E2 -451.323} C_VEL
LIN {X 0,Y 608.441,Z 862.203,A -85,B 0,C 180,E1 -451.985,E2 -451.985} C_VEL
LIN {X 0,Y 608.425,Z 860.811,A -85,B 0,C 180,E1 -452.648,E2 -452.648} C_VEL
LIN {X 0,Y 608.449,Z 857.899,A -85,B 0,C 180,E1 -453.642,E2 -453.642} C_VEL
LIN {X 0,Y 608.432,Z 853.953,A -85,B 0,C 180,E1 -454.637,E2 -454.637} C_VEL
LIN {X 0,Y 608.437,Z 847.881,A -85,B 0,C 180,E1 -455.8,E2 -455.8} C_VEL
LIN {X 0,Y 608.461,Z 841.241,A -85,B 0,C 180,E1 -456.799,E2 -456.799} C_VEL
LIN {X 0,Y 608.455,Z 832.996,A -85,B 0,C 180,E1 -457.799,E2 -457.799} C_VEL
LIN {X 0,Y 608.472,Z 824.545,A -85,B 0,C 180,E1 -458.635,E2 -458.635} C_VEL
LIN {X 0,Y 608.471,Z 814.102,A -85,B 0,C 180,E1 -459.473,E2 -459.473} C_VEL
LIN {X 0,Y 608.487,Z 803.769,A -85,B 0,C 180,E1 -460.144,E2 -460.144} C_VEL
LIN {X 0,Y 608.521,Z 792.258,A -85,B 0,C 180,E1 -460.74,E2 -460.74} C_VEL
LIN {X 0,Y 608.532,Z 780.897,A -85,B 0,C 180,E1 -461.192,E2 -461.192} C_VEL
LIN {X 0,Y 608.535,Z 768.301,A -85,B 0,C 180,E1 -461.554,E2 -461.554} C_VEL
LIN {X 0,Y 608.53,Z 755.659,A -85,B 0,C 180,E1 -461.786,E2 -461.786} C_VEL
LIN {X 0,Y 608.467,Z 651.276,A -85,B 0,C 180,E1 -463.037,E2 -463.037} C_VEL
LIN {X 0,Y 608.489,Z 630.975,A -85,B 0,C 180,E1 -465.576,E2 -465.576} C_VEL
LIN {X 0,Y 608.544,Z 609.227,A -85,B 0,C 180,E1 -468.331,E2 -468.331} C_VEL
LIN {X 0,Y 608.57,Z 587.304,A -85,B 0,C 180,E1 -471.154,E2 -471.154} C_VEL
LIN {X 0,Y 608.524,Z 569.903,A -85,B 0,C 180,E1 -473.435,E2 -473.435} C_VEL
LIN {X 0,Y 608.46,Z 569.689,A -85,B 0,C 180,E1 -473.844,E2 -473.844} C_VEL
LIN {X 0,Y 608.45,Z 569.695,A -85,B 0,C 180,E1 -476.773,E2 -476.773} C_VEL
LIN {X 0,Y 608.474,Z 569.688,A -85,B 0,C 180,E1 -479.019,E2 -479.019} C_VEL
LIN {X 0,Y 608.444,Z 569.689,A -85,B 0,C 180,E1 -481.317,E2 -481.317} C_VEL
LIN {X 0,Y 608.475,Z 569.685,A -85,B 0,C 180,E1 -483.735,E2 -483.735} C_VEL
LIN {X 0,Y 608.474,Z 569.688,A -85,B 0,C 180,E1 -486.089,E2 -486.089} C_VEL
LIN {X 0,Y 608.464,Z 569.696,A -85,B 0,C 180,E1 -488.587,E2 -488.587} C_VEL
LIN {X 0,Y 608.455,Z 569.687,A -85,B 0,C 180,E1 -491.341,E2 -491.341} C_VEL
LIN {X 0,Y 608.452,Z 569.694,A -85,B 0,C 180,E1 -494.263,E2 -494.263} C_VEL
LIN {X 0,Y 608.452,Z 569.689,A -85,B 0,C 180,E1 -497.04,E2 -497.04} C_VEL
LIN {X 0,Y 608.453,Z 569.688,A -85,B 0,C 180,E1 -499.696,E2 -499.696} C_VEL
LIN {X 0,Y 608.474,Z 569.692,A -85,B 0,C 180,E1 -502.254,E2 -502.254} C_VEL
LIN {X 0,Y 608.47,Z 569.686,A -85,B 0,C 180,E1 -505.09,E2 -505.09} C_VEL
LIN {X 0,Y 608.464,Z 569.688,A -85,B 0,C 180,E1 -507.905,E2 -507.905} C_VEL
LIN {X 0,Y 608.479,Z 569.691,A -85,B 0,C 180,E1 -510.221,E2 -510.221} C_VEL
LIN {X 0,Y 608.446,Z 569.688,A -85,B 0,C 180,E1 -513.225,E2 -513.225} C_VEL
LIN {X 0,Y 608.475,Z 569.686,A -85,B 0,C 180,E1 -515.846,E2 -515.846} C_VEL
LIN {X 0,Y 608.46,Z 569.696,A -85,B 0,C 180,E1 -518.308,E2 -518.308} C_VEL
LIN {X 0,Y 608.45,Z 569.688,A -85,B 0,C 180,E1 -521.13,E2 -521.13} C_VEL
LIN {X 0,Y 608.456,Z 569.69,A -85,B 0,C 180,E1 -523.906,E2 -523.906} C_VEL
LIN {X 0,Y 608.456,Z 569.693,A -85,B 0,C 180,E1 -526.643,E2 -526.643} C_VEL
LIN {X 0,Y 608.462,Z 569.686,A -85,B 0,C 180,E1 -529.35,E2 -529.35} C_VEL
LIN {X 0,Y 608.474,Z 569.69,A -85,B 0,C 180,E1 -532.033,E2 -532.033} C_VEL
LIN {X 0,Y 608.457,Z 569.691,A -85,B 0,C 180,E1 -534.698,E2 -534.698} C_VEL
LIN {X 0,Y 608.483,Z 569.683,A -85,B 0,C 180,E1 -537.352,E2 -537.352} C_VEL
LIN {X 0,Y 608.469,Z 569.69,A -85,B 0,C 180,E1 -540,E2 -540} C_VEL
LIN {X 0,Y 608.483,Z 569.688,A -85,B 0,C 180,E1 -542.648,E2 -542.648} C_VEL
LIN {X 0,Y 608.458,Z 569.686,A -85,B 0,C 180,E1 -545.302,E2 -545.302} C_VEL
LIN {X 0,Y 608.475,Z 569.69,A -85,B 0,C 180,E1 -547.967,E2 -547.967} C_VEL
LIN {X 0,Y 608.452,Z 569.688,A -85,B 0,C 180,E1 -549.471,E2 -549.471} C_VEL
LIN {X 0,Y 607.779,Z 569.779,A -85,B 0,C 180,E1 -550.024,E2 -550.024} C_VEL
LIN {X 0,Y 604.927,Z 570.136,A -85,B 0,C 180,E1 -550.921,E2 -550.921} C_VEL
LIN {X 0,Y 602.523,Z 570.436,A -85,B 0,C 180,E1 -551.642,E2 -551.642} C_VEL
LIN {X 0,Y 601.493,Z 570.564,A -85,B 0,C 180,E1 -552.199,E2 -552.199} C_VEL
LIN {X 0,Y 601.41,Z 570.57,A -85,B 0,C 180,E1 -552.388,E2 -552.388} C_VEL
LIN {X 0,Y 601.427,Z 570.565,A -85,B 0,C 180,E1 -554.897,E2 -554.897} C_VEL
LIN {X 0,Y 601.433,Z 570.564,A -85,B 0,C 180,E1 -557.599,E2 -557.599} C_VEL
LIN {X 0,Y 601.423,Z 584.448,A -85,B 0,C 180,E1 -560.165,E2 -560.165} C_VEL
LIN {X 0,Y 601.42,Z 593.885,A -85,B 0,C 180,E1 -561.891,E2 -561.891} C_VEL
LIN {X 0,Y 601.657,Z 601.784,A -85,B 0,C 180,E1 -561.994,E2 -561.994} C_VEL
LIN {X 0,Y 601.589,Z 700.711,A -85,B 0,C 180,E1 -563.198,E2 -563.198} C_VEL
LIN {X 0,Y 601.574,Z 713.643,A -85,B 0,C 180,E1 -563.495,E2 -563.495} C_VEL
LIN {X 0,Y 601.55,Z 725.879,A -85,B 0,C 180,E1 -563.907,E2 -563.907} C_VEL
LIN {X 0,Y 601.514,Z 738.17,A -85,B 0,C 180,E1 -564.469,E2 -564.469} C_VEL
LIN {X 0,Y 601.457,Z 749.695,A -85,B 0,C 180,E1 -565.153,E2 -565.153} C_VEL
LIN {X 0,Y 601.45,Z 760.185,A -85,B 0,C 180,E1 -565.931,E2 -565.931} C_VEL
LIN {X 0,Y 601.404,Z 769.051,A -85,B 0,C 180,E1 -566.738,E2 -566.738} C_VEL
LIN {X 0,Y 601.386,Z 777.883,A -85,B 0,C 180,E1 -567.727,E2 -567.727} C_VEL
LIN {X 0,Y 601.373,Z 785.467,A -85,B 0,C 180,E1 -568.78,E2 -568.78} C_VEL
LIN {X 0,Y 601.376,Z 791.135,A -85,B 0,C 180,E1 -569.765,E2 -569.765} C_VEL
LIN {X 0,Y 601.333,Z 796.395,A -85,B 0,C 180,E1 -570.947,E2 -570.947} C_VEL
LIN {X 0,Y 601.329,Z 800.179,A -85,B 0,C 180,E1 -572.126,E2 -572.126} C_VEL
LIN {X 0,Y 601.324,Z 802.668,A -85,B 0,C 180,E1 -573.32,E2 -573.32} C_VEL
LIN {X 0,Y 601.318,Z 803.61,A -85,B 0,C 180,E1 -574.125,E2 -574.125} C_VEL
LIN {X 0,Y 601.317,Z 803.993,A -85,B 0,C 180,E1 -575.103,E2 -575.103} C_VEL
LIN {X 0,Y 601.335,Z 803.336,A -85,B 0,C 180,E1 -576.254,E2 -576.254} C_VEL
LIN {X 0,Y 601.326,Z 801.458,A -85,B 0,C 180,E1 -577.427,E2 -577.427} C_VEL
LIN {X 0,Y 601.324,Z 798.754,A -85,B 0,C 180,E1 -578.46,E2 -578.46} C_VEL
LIN {X 0,Y 601.363,Z 793.943,A -85,B 0,C 180,E1 -579.74,E2 -579.74} C_VEL
LIN {X 0,Y 601.348,Z 788.087,A -85,B 0,C 180,E1 -580.88,E2 -580.88} C_VEL
LIN {X 0,Y 601.369,Z 780.874,A -85,B 0,C 180,E1 -581.975,E2 -581.975} C_VEL
LIN {X 0,Y 601.415,Z 772.308,A -85,B 0,C 180,E1 -583.012,E2 -583.012} C_VEL
LIN {X 0,Y 601.457,Z 762.837,A -85,B 0,C 180,E1 -583.931,E2 -583.931} C_VEL
LIN {X 0,Y 601.472,Z 752.471,A -85,B 0,C 180,E1 -584.748,E2 -584.748} C_VEL
LIN {X 0,Y 601.48,Z 741.145,A -85,B 0,C 180,E1 -585.46,E2 -585.46} C_VEL
LIN {X 0,Y 601.525,Z 728.467,A -85,B 0,C 180,E1 -586.077,E2 -586.077} C_VEL
LIN {X 0,Y 601.57,Z 715.496,A -85,B 0,C 180,E1 -586.543,E2 -586.543} C_VEL
LIN {X 0,Y 601.604,Z 702.253,A -85,B 0,C 180,E1 -586.863,E2 -586.863} C_VEL
LIN {X 0,Y 601.599,Z 680.976,A -85,B 0,C 180,E1 -587.148,E2 -587.148} C_VEL
LIN {X 0,Y 601.494,Z 594.562,A -85,B 0,C 180,E1 -588.186,E2 -588.186} C_VEL
LIN {X 0,Y 601.411,Z 593.687,A -85,B 0,C 180,E1 -588.235,E2 -588.235} C_VEL
LIN {X 0,Y 601.441,Z 579.274,A -85,B 0,C 180,E1 -590.877,E2 -590.877} C_VEL
LIN {X 0,Y 601.445,Z 570.562,A -85,B 0,C 180,E1 -592.53,E2 -592.53} C_VEL
LIN {X 0,Y 601.433,Z 570.562,A -85,B 0,C 180,E1 -595.07,E2 -595.07} C_VEL
LIN {X 0,Y 601.433,Z 570.565,A -85,B 0,C 180,E1 -597.485,E2 -597.485} C_VEL
LIN {X 0,Y 601.426,Z 570.571,A -85,B 0,C 180,E1 -599.852,E2 -599.852} C_VEL
LIN {X 0,Y 601.413,Z 570.565,A -85,B 0,C 180,E1 -602.638,E2 -602.638} C_VEL
LIN {X 0,Y 601.4,Z 570.565,A -85,B 0,C 180,E1 -605.122,E2 -605.122} C_VEL
LIN {X 0,Y 601.414,Z 570.564,A -85,B 0,C 180,E1 -607.395,E2 -607.395} C_VEL
LIN {X 0,Y 601.409,Z 570.576,A -85,B 0,C 180,E1 -610.192,E2 -610.192} C_VEL
LIN {X 0,Y 601.433,Z 570.562,A -85,B 0,C 180,E1 -613.015,E2 -613.015} C_VEL
LIN {X 0,Y 601.422,Z 570.567,A -85,B 0,C 180,E1 -615.909,E2 -615.909} C_VEL
LIN {X 0,Y 601.44,Z 570.568,A -85,B 0,C 180,E1 -618.543,E2 -618.543} C_VEL
LIN {X 0,Y 601.413,Z 570.564,A -85,B 0,C 180,E1 -621.263,E2 -621.263} C_VEL
LIN {X 0,Y 601.416,Z 570.566,A -85,B 0,C 180,E1 -623.964,E2 -623.964} C_VEL
LIN {X 0,Y 601.435,Z 570.569,A -85,B 0,C 180,E1 -626.651,E2 -626.651} C_VEL
LIN {X 0,Y 601.442,Z 570.56,A -85,B 0,C 180,E1 -629.331,E2 -629.331} C_VEL
LIN {X 0,Y 601.434,Z 570.563,A -85,B 0,C 180,E1 -632.01,E2 -632.01} C_VEL
LIN {X 0,Y 601.43,Z 570.572,A -85,B 0,C 180,E1 -634.693,E2 -634.693} C_VEL
LIN {X 0,Y 601.443,Z 570.561,A -85,B 0,C 180,E1 -637.386,E2 -637.386} C_VEL
LIN {X 0,Y 601.432,Z 570.563,A -85,B 0,C 180,E1 -640.096,E2 -640.096} C_VEL
LIN {X 0,Y 601.428,Z 570.572,A -85,B 0,C 180,E1 -642.829,E2 -642.829} C_VEL
LIN {X 0,Y 601.413,Z 570.564,A -85,B 0,C 180,E1 -645.592,E2 -645.592} C_VEL
LIN {X 0,Y 601.401,Z 570.565,A -85,B 0,C 180,E1 -647.689,E2 -647.689} C_VEL
LIN {X 0,Y 601.435,Z 570.565,A -85,B 0,C 180,E1 -650.522,E2 -650.522} C_VEL
LIN {X 0,Y 601.398,Z 570.569,A -85,B 0,C 180,E1 -653.412,E2 -653.412} C_VEL
LIN {X 0,Y 601.412,Z 570.564,A -85,B 0,C 180,E1 -655.867,E2 -655.867} C_VEL
LIN {X 0,Y 601.407,Z 570.565,A -85,B 0,C 180,E1 -657.869,E2 -657.869} C_VEL
LIN {X 0,Y 601.431,Z 570.561,A -85,B 0,C 180,E1 -660.165,E2 -660.165} C_VEL
LIN {X 0,Y 601.423,Z 570.566,A -85,B 0,C 180,E1 -662.715,E2 -662.715} C_VEL
LIN {X 0,Y 601.418,Z 570.573,A -85,B 0,C 180,E1 -665.115,E2 -665.115} C_VEL
LIN {X 0,Y 601.439,Z 570.568,A -85,B 0,C 180,E1 -667.419,E2 -667.419} C_VEL
LIN {X 0,Y 601.415,Z 570.564,A -85,B 0,C 180,E1 -669.995,E2 -669.995} C_VEL
LIN {X 0,Y 601.413,Z 570.565,A -85,B 0,C 180,E1 -672.671,E2 -672.671} C_VEL
LIN {X 0,Y 601.431,Z 570.571,A -85,B 0,C 180,E1 -675.482,E2 -675.482} C_VEL
LIN {X 0,Y 601.426,Z 570.562,A -85,B 0,C 180,E1 -678.407,E2 -678.407} C_VEL
LIN {X 0,Y 601.44,Z 570.571,A -85,B 0,C 180,E1 -681.529,E2 -681.529} C_VEL
LIN {X 0,Y 601.389,Z 570.568,A -85,B 0,C 180,E1 -684.245,E2 -684.245} C_VEL
LIN {X 0,Y 601.421,Z 570.563,A -85,B 0,C 180,E1 -686.686,E2 -686.686} C_VEL
LIN {X 0,Y 601.418,Z 570.565,A -85,B 0,C 180,E1 -689.058,E2 -689.058} C_VEL
LIN {X 0,Y 601.438,Z 570.566,A -85,B 0,C 180,E1 -691.374,E2 -691.374} C_VEL
LIN {X 0,Y 601.407,Z 570.574,A -85,B 0,C 180,E1 -693.636,E2 -693.636} C_VEL
LIN {X 0,Y 601.457,Z 570.567,A -85,B 0,C 180,E1 -695.86,E2 -695.86} C_VEL
LIN {X 0,Y 601.408,Z 570.564,A -85,B 0,C 180,E1 -698.761,E2 -698.761} C_VEL
LIN {X 0,Y 601.424,Z 570.569,A -85,B 0,C 180,E1 -701.608,E2 -701.608} C_VEL
LIN {X 0,Y 601.443,Z 570.568,A -85,B 0,C 180,E1 -703.713,E2 -703.713} C_VEL
LIN {X 0,Y 601.415,Z 570.566,A -85,B 0,C 180,E1 -706.484,E2 -706.484} C_VEL
LIN {X 0,Y 601.421,Z 570.563,A -85,B 0,C 180,E1 -709.224,E2 -709.224} C_VEL
LIN {X 0,Y 601.447,Z 570.569,A -85,B 0,C 180,E1 -711.939,E2 -711.939} C_VEL
LIN {X 0,Y 601.425,Z 570.564,A -85,B 0,C 180,E1 -714.636,E2 -714.636} C_VEL
LIN {X 0,Y 601.449,Z 570.559,A -85,B 0,C 180,E1 -717.321,E2 -717.321} C_VEL
LIN {X 0,Y 601.45,Z 570.567,A -85,B 0,C 180,E1 -720,E2 -720} C_VEL
LIN {X 0,Y 601.449,Z 570.563,A -85,B 0,C 180,E1 -722.679,E2 -722.679} C_VEL
LIN {X 0,Y 601.423,Z 570.562,A -85,B 0,C 180,E1 -725.364,E2 -725.364} C_VEL
LIN {X 0,Y 601.446,Z 570.566,A -85,B 0,C 180,E1 -728.061,E2 -728.061} C_VEL
LIN {X 0,Y 601.43,Z 570.563,A -85,B 0,C 180,E1 -731.012,E2 -731.012} C_VEL
LIN {X 0,Y 601.416,Z 570.563,A -85,B 0,C 180,E1 -733.516,E2 -733.516} C_VEL
LIN {X 0,Y 601.443,Z 570.567,A -85,B 0,C 180,E1 -736.287,E2 -736.287} C_VEL
LIN {X 0,Y 601.421,Z 570.565,A -85,B 0,C 180,E1 -739.099,E2 -739.099} C_VEL
LIN {X 0,Y 601.408,Z 570.565,A -85,B 0,C 180,E1 -741.239,E2 -741.239} C_VEL
LIN {X 0,Y 601.461,Z 570.561,A -85,B 0,C 180,E1 -744.14,E2 -744.14} C_VEL
LIN {X 0,Y 601.45,Z 570.563,A -85,B 0,C 180,E1 -747.111,E2 -747.111} C_VEL
LIN {X 0,Y 601.42,Z 570.564,A -85,B 0,C 180,E1 -749.393,E2 -749.393} C_VEL
LIN {X 0,Y 601.404,Z 570.565,A -85,B 0,C 180,E1 -751.727,E2 -751.727} C_VEL
LIN {X 0,Y 601.436,Z 570.562,A -85,B 0,C 180,E1 -754.118,E2 -754.118} C_VEL
LIN {X 0,Y 601.441,Z 570.563,A -85,B 0,C 180,E1 -757.382,E2 -757.382} C_VEL
LIN {X 0,Y 601.406,Z 570.564,A -85,B 0,C 180,E1 -759.996,E2 -759.996} C_VEL
LIN {X 0,Y 601.419,Z 570.569,A -85,B 0,C 180,E1 -762.67,E2 -762.67} C_VEL
LIN {X 0,Y 601.403,Z 570.568,A -85,B 0,C 180,E1 -765.479,E2 -765.479} C_VEL
LIN {X 0,Y 601.425,Z 570.563,A -85,B 0,C 180,E1 -768.407,E2 -768.407} C_VEL
LIN {X 0,Y 601.434,Z 570.568,A -85,B 0,C 180,E1 -770.875,E2 -770.875} C_VEL
LIN {X 0,Y 601.406,Z 570.571,A -85,B 0,C 180,E1 -773.417,E2 -773.417} C_VEL
LIN {X 0,Y 601.438,Z 570.561,A -85,B 0,C 180,E1 -776.064,E2 -776.064} C_VEL
LIN {X 0,Y 601.424,Z 570.563,A -85,B 0,C 180,E1 -778.545,E2 -778.545} C_VEL
LIN {X 0,Y 601.44,Z 570.571,A -85,B 0,C 180,E1 -781.373,E2 -781.373} C_VEL
LIN {X 0,Y 601.405,Z 570.571,A -85,B 0,C 180,E1 -783.636,E2 -783.636} C_VEL
LIN {X 0,Y 601.433,Z 570.574,A -85,B 0,C 180,E1 -786.361,E2 -786.361} C_VEL
LIN {X 0,Y 601.729,Z 575.009,A -85,B 0,C 180,E1 -786.966,E2 -786.966} C_VEL
LIN {X 0,Y 601.621,Z 596.845,A -85,B 0,C 180,E1 -789.841,E2 -789.841} C_VEL
LIN {X 0,Y 601.558,Z 618.681,A -85,B 0,C 180,E1 -792.667,E2 -792.667} C_VEL
LIN {X 0,Y 601.504,Z 641.882,A -85,B 0,C 180,E1 -795.623,E2 -795.623} C_VEL
LIN {X 0,Y 601.457,Z 651.349,A -85,B 0,C 180,E1 -796.818,E2 -796.818} C_VEL
LIN {X 0,Y 601.634,Z 671.763,A -85,B 0,C 180,E1 -797.069,E2 -797.069} C_VEL
LIN {X 0,Y 601.599,Z 759.911,A -85,B 0,C 180,E1 -798.139,E2 -798.139} C_VEL
LIN {X 0,Y 601.58,Z 773.193,A -85,B 0,C 180,E1 -798.437,E2 -798.437} C_VEL
LIN {X 0,Y 601.549,Z 784.915,A -85,B 0,C 180,E1 -798.826,E2 -798.826} C_VEL
LIN {X 0,Y 601.516,Z 795.909,A -85,B 0,C 180,E1 -799.31,E2 -799.31} C_VEL
LIN {X 0,Y 601.471,Z 806.569,A -85,B 0,C 180,E1 -799.905,E2 -799.905} C_VEL
LIN {X 0,Y 601.446,Z 817.467,A -85,B 0,C 180,E1 -800.669,E2 -800.669} C_VEL
LIN {X 0,Y 601.429,Z 828.105,A -85,B 0,C 180,E1 -801.6,E2 -801.6} C_VEL
LIN {X 0,Y 601.418,Z 835.955,A -85,B 0,C 180,E1 -802.445,E2 -802.445} C_VEL
LIN {X 0,Y 601.371,Z 843.221,A -85,B 0,C 180,E1 -803.397,E2 -803.397} C_VEL
LIN {X 0,Y 601.372,Z 848.862,A -85,B 0,C 180,E1 -804.298,E2 -804.298} C_VEL
LIN {X 0,Y 601.336,Z 853.947,A -85,B 0,C 180,E1 -805.307,E2 -805.307} C_VEL
LIN {X 0,Y 601.368,Z 857.894,A -85,B 0,C 180,E1 -806.314,E2 -806.314} C_VEL
LIN {X 0,Y 601.325,Z 860.807,A -85,B 0,C 180,E1 -807.32,E2 -807.32} C_VEL
LIN {X 0,Y 601.34,Z 862.2,A -85,B 0,C 180,E1 -807.99,E2 -807.99} C_VEL
LIN {X 0,Y 601.339,Z 863.783,A -85,B 0,C 180,E1 -809.33,E2 -809.33} C_VEL
LIN {X 0,Y 601.335,Z 864,A -85,B 0,C 180,E1 -809.999,E2 -809.999} C_VEL
LIN {X 0,Y 601.348,Z 863.185,A -85,B 0,C 180,E1 -811.339,E2 -811.339} C_VEL
LIN {X 0,Y 601.34,Z 862.203,A -85,B 0,C 180,E1 -812.009,E2 -812.009} C_VEL
LIN {X 0,Y 601.325,Z 860.811,A -85,B 0,C 180,E1 -812.679,E2 -812.679} C_VEL
LIN {X 0,Y 601.368,Z 857.899,A -85,B 0,C 180,E1 -813.685,E2 -813.685} C_VEL
LIN {X 0,Y 601.336,Z 853.953,A -85,B 0,C 180,E1 -814.692,E2 -814.692} C_VEL
LIN {X 0,Y 601.372,Z 847.881,A -85,B 0,C 180,E1 -815.868,E2 -815.868} C_VEL
LIN {X 0,Y 601.387,Z 841.241,A -85,B 0,C 180,E1 -816.879,E2 -816.879} C_VEL
LIN {X 0,Y 601.4,Z 832.996,A -85,B 0,C 180,E1 -817.892,E2 -817.892} C_VEL
LIN {X 0,Y 601.436,Z 824.545,A -85,B 0,C 180,E1 -818.737,E2 -818.737} C_VEL
LIN {X 0,Y 601.44,Z 814.103,A -85,B 0,C 180,E1 -819.584,E2 -819.584} C_VEL
LIN {X 0,Y 601.489,Z 803.77,A -85,B 0,C 180,E1 -820.263,E2 -820.263} C_VEL
LIN {X 0,Y 601.536,Z 792.913,A -85,B 0,C 180,E1 -820.835,E2 -820.835} C_VEL
LIN {X 0,Y 601.565,Z 780.398,A -85,B 0,C 180,E1 -821.34,E2 -821.34} C_VEL
LIN {X 0,Y 601.593,Z 767.387,A -85,B 0,C 180,E1 -821.71,E2 -821.71} C_VEL
LIN {X 0,Y 601.606,Z 754.146,A -85,B 0,C 180,E1 -821.945,E2 -821.945} C_VEL
LIN {X 0,Y 601.565,Z 652.211,A -85,B 0,C 180,E1 -823.168,E2 -823.168} C_VEL
LIN {X 0,Y 601.462,Z 651.276,A -85,B 0,C 180,E1 -823.191,E2 -823.191} C_VEL
LIN {X 0,Y 601.512,Z 629.611,A -85,B 0,C 180,E1 -825.936,E2 -825.936} C_VEL
LIN {X 0,Y 601.605,Z 608.662,A -85,B 0,C 180,E1 -828.623,E2 -828.623} C_VEL
LIN {X 0,Y 601.676,Z 585.939,A -85,B 0,C 180,E1 -831.588,E2 -831.588} C_VEL
LIN {X 0,Y 601.752,Z 572.292,A -85,B 0,C 180,E1 -833.396,E2 -833.396} C_VEL
LIN {X 0,Y 601.423,Z 570.567,A -85,B 0,C 180,E1 -833.66,E2 -833.66} C_VEL
LIN {X 0,Y 601.403,Z 570.573,A -85,B 0,C 180,E1 -836.363,E2 -836.363} C_VEL
LIN {X 0,Y 601.442,Z 570.567,A -85,B 0,C 180,E1 -838.789,E2 -838.789} C_VEL
LIN {X 0,Y 601.401,Z 570.566,A -85,B 0,C 180,E1 -841.726,E2 -841.726} C_VEL
LIN {X 0,Y 601.43,Z 570.566,A -85,B 0,C 180,E1 -844.117,E2 -844.117} C_VEL
LIN {X 0,Y 601.408,Z 570.575,A -85,B 0,C 180,E1 -846.581,E2 -846.581} C_VEL
LIN {X 0,Y 601.438,Z 570.561,A -85,B 0,C 180,E1 -849.535,E2 -849.535} C_VEL
LIN {X 0,Y 601.41,Z 570.574,A -85,B 0,C 180,E1 -852.59,E2 -852.59} C_VEL
LIN {X 0,Y 601.421,Z 570.563,A -85,B 0,C 180,E1 -855.481,E2 -855.481} C_VEL
LIN {X 0,Y 601.425,Z 570.572,A -85,B 0,C 180,E1 -858.405,E2 -858.405} C_VEL
LIN {X 0,Y 601.436,Z 570.565,A -85,B 0,C 180,E1 -860.875,E2 -860.875} C_VEL
LIN {X 0,Y 601.439,Z 570.562,A -85,B 0,C 180,E1 -863.733,E2 -863.733} C_VEL
LIN {X 0,Y 601.428,Z 570.569,A -85,B 0,C 180,E1 -866.686,E2 -866.686} C_VEL
LIN {X 0,Y 601.427,Z 570.564,A -85,B 0,C 180,E1 -869.058,E2 -869.058} C_VEL
LIN {X 0,Y 601.425,Z 570.562,A -85,B 0,C 180,E1 -871.373,E2 -871.373} C_VEL
LIN {X 0,Y 601.417,Z 570.569,A -85,B 0,C 180,E1 -874.13,E2 -874.13} C_VEL
LIN {X 0,Y 601.418,Z 570.571,A -85,B 0,C 180,E1 -876.589,E2 -876.589} C_VEL
LIN {X 0,Y 601.427,Z 570.562,A -85,B 0,C 180,E1 -879.478,E2 -879.478} C_VEL
LIN {X 0,Y 601.393,Z 570.576,A -85,B 0,C 180,E1 -882.311,E2 -882.311} C_VEL
LIN {X 0,Y 601.409,Z 570.575,A -85,B 0,C 180,E1 -884.408,E2 -884.408} C_VEL
LIN {X 0,Y 601.417,Z 570.564,A -85,B 0,C 180,E1 -887.172,E2 -887.172} C_VEL
LIN {X 0,Y 601.431,Z 570.565,A -85,B 0,C 180,E1 -889.905,E2 -889.905} C_VEL
LIN {X 0,Y 601.433,Z 570.568,A -85,B 0,C 180,E1 -892.615,E2 -892.615} C_VEL
LIN {X 0,Y 601.431,Z 570.562,A -85,B 0,C 180,E1 -895.308,E2 -895.308} C_VEL
LIN {X 0,Y 601.417,Z 570.569,A -85,B 0,C 180,E1 -897.991,E2 -897.991} C_VEL
LIN {X 0,Y 601.447,Z 570.565,A -85,B 0,C 180,E1 -900.669,E2 -900.669} C_VEL
LIN {X 0,Y 601.425,Z 570.563,A -85,B 0,C 180,E1 -903.349,E2 -903.349} C_VEL
LIN {X 0,Y 601.431,Z 570.568,A -85,B 0,C 180,E1 -906.037,E2 -906.037} C_VEL
LIN {X 0,Y 601.439,Z 570.564,A -85,B 0,C 180,E1 -908.737,E2 -908.737} C_VEL
LIN {X 0,Y 601.428,Z 570.563,A -85,B 0,C 180,E1 -911.458,E2 -911.458} C_VEL
LIN {X 0,Y 601.41,Z 570.57,A -85,B 0,C 180,E1 -912.388,E2 -912.388} C_VEL
LIN {X 0,Y 600.745,Z 570.65,A -85,B 0,C 180,E1 -912.947,E2 -912.947} C_VEL
LIN {X 0,Y 597.893,Z 571.007,A -85,B 0,C 180,E1 -913.855,E2 -913.855} C_VEL
LIN {X 0,Y 595.481,Z 571.309,A -85,B 0,C 180,E1 -914.585,E2 -914.585} C_VEL
LIN {X 0,Y 594.443,Z 571.434,A -85,B 0,C 180,E1 -915.148,E2 -915.148} C_VEL
LIN {X 0,Y 594.358,Z 571.444,A -85,B 0,C 180,E1 -915.339,E2 -915.339} C_VEL
LIN {X 0,Y 594.401,Z 571.54,A -85,B 0,C 180,E1 -917.57,E2 -917.57} C_VEL
LIN {X 0,Y 594.389,Z 584.816,A -85,B 0,C 180,E1 -920.053,E2 -920.053} C_VEL
LIN {X 0,Y 594.39,Z 593.87,A -85,B 0,C 180,E1 -921.73,E2 -921.73} C_VEL
LIN {X 0,Y 594.749,Z 599.102,A -85,B 0,C 180,E1 -921.807,E2 -921.807} C_VEL
LIN {X 0,Y 594.642,Z 700.175,A -85,B 0,C 180,E1 -923.048,E2 -923.048} C_VEL
LIN {X 0,Y 594.62,Z 713.284,A -85,B 0,C 180,E1 -923.348,E2 -923.348} C_VEL
LIN {X 0,Y 594.569,Z 726.247,A -85,B 0,C 180,E1 -923.789,E2 -923.789} C_VEL
LIN {X 0,Y 594.533,Z 738.787,A -85,B 0,C 180,E1 -924.378,E2 -924.378} C_VEL
LIN {X 0,Y 594.448,Z 750.465,A -85,B 0,C 180,E1 -925.087,E2 -925.087} C_VEL
LIN {X 0,Y 594.404,Z 760.501,A -85,B 0,C 180,E1 -925.849,E2 -925.849} C_VEL
LIN {X 0,Y 594.339,Z 769.658,A -85,B 0,C 180,E1 -926.702,E2 -926.702} C_VEL
LIN {X 0,Y 594.326,Z 777.847,A -85,B 0,C 180,E1 -927.635,E2 -927.635} C_VEL
LIN {X 0,Y 594.3,Z 784.695,A -85,B 0,C 180,E1 -928.587,E2 -928.587} C_VEL
LIN {X 0,Y 594.283,Z 790.526,A -85,B 0,C 180,E1 -929.586,E2 -929.586} C_VEL
LIN {X 0,Y 594.286,Z 795.076,A -85,B 0,C 180,E1 -930.565,E2 -930.565} C_VEL
LIN {X 0,Y 594.244,Z 798.861,A -85,B 0,C 180,E1 -931.624,E2 -931.624} C_VEL
LIN {X 0,Y 594.242,Z 802.116,A -85,B 0,C 180,E1 -932.959,E2 -932.959} C_VEL
LIN {X 0,Y 594.242,Z 803.614,A -85,B 0,C 180,E1 -934.121,E2 -934.121} C_VEL
LIN {X 0,Y 594.223,Z 803.921,A -85,B 0,C 180,E1 -935.418,E2 -935.418} C_VEL
LIN {X 0,Y 594.233,Z 803.109,A -85,B 0,C 180,E1 -936.465,E2 -936.465} C_VEL
LIN {X 0,Y 594.23,Z 801.174,A -85,B 0,C 180,E1 -937.59,E2 -937.59} C_VEL
LIN {X 0,Y 594.247,Z 797.756,A -85,B 0,C 180,E1 -938.816,E2 -938.816} C_VEL
LIN {X 0,Y 594.282,Z 792.321,A -85,B 0,C 180,E1 -940.144,E2 -940.144} C_VEL
LIN {X 0,Y 594.288,Z 786.044,A -85,B 0,C 180,E1 -941.293,E2 -941.293} C_VEL
LIN {X 0,Y 594.309,Z 778.44,A -85,B 0,C 180,E1 -942.381,E2 -942.381} C_VEL
LIN {X 0,Y 594.359,Z 769.198,A -85,B 0,C 180,E1 -943.436,E2 -943.436} C_VEL
LIN {X 0,Y 594.411,Z 760.594,A -85,B 0,C 180,E1 -944.233,E2 -944.233} C_VEL
LIN {X 0,Y 594.454,Z 750.95,A -85,B 0,C 180,E1 -944.97,E2 -944.97} C_VEL
LIN {X 0,Y 594.498,Z 738.986,A -85,B 0,C 180,E1 -945.702,E2 -945.702} C_VEL
LIN {X 0,Y 594.586,Z 726.734,A -85,B 0,C 180,E1 -946.281,E2 -946.281} C_VEL
LIN {X 0,Y 594.642,Z 713.823,A -85,B 0,C 180,E1 -946.727,E2 -946.727} C_VEL
LIN {X 0,Y 594.642,Z 700.679,A -85,B 0,C 180,E1 -947.033,E2 -947.033} C_VEL
LIN {X 0,Y 594.615,Z 595.379,A -85,B 0,C 180,E1 -948.331,E2 -948.331} C_VEL
LIN {X 0,Y 594.374,Z 593.806,A -85,B 0,C 180,E1 -948.372,E2 -948.372} C_VEL
LIN {X 0,Y 594.404,Z 578.076,A -85,B 0,C 180,E1 -951.293,E2 -951.293} C_VEL
LIN {X 0,Y 594.416,Z 571.438,A -85,B 0,C 180,E1 -952.55,E2 -952.55} C_VEL
LIN {X 0,Y 594.394,Z 571.442,A -85,B 0,C 180,E1 -955.422,E2 -955.422} C_VEL
LIN {X 0,Y 594.376,Z 571.445,A -85,B 0,C 180,E1 -958.358,E2 -958.358} C_VEL
LIN {X 0,Y 594.382,Z 571.439,A -85,B 0,C 180,E1 -961.043,E2 -961.043} C_VEL
LIN {X 0,Y 594.385,Z 571.449,A -85,B 0,C 180,E1 -963.978,E2 -963.978} C_VEL
LIN {X 0,Y 594.39,Z 571.446,A -85,B 0,C 180,E1 -966.297,E2 -966.297} C_VEL
LIN {X 0,Y 594.402,Z 571.437,A -85,B 0,C 180,E1 -969.225,E2 -969.225} C_VEL
LIN {X 0,Y 594.383,Z 571.448,A -85,B 0,C 180,E1 -972.097,E2 -972.097} C_VEL
LIN {X 0,Y 594.371,Z 571.452,A -85,B 0,C 180,E1 -974.22,E2 -974.22} C_VEL
LIN {X 0,Y 594.369,Z 571.442,A -85,B 0,C 180,E1 -977.018,E2 -977.018} C_VEL
LIN {X 0,Y 594.393,Z 571.44,A -85,B 0,C 180,E1 -979.785,E2 -979.785} C_VEL
LIN {X 0,Y 594.397,Z 571.447,A -85,B 0,C 180,E1 -982.528,E2 -982.528} C_VEL
LIN {X 0,Y 594.387,Z 571.439,A -85,B 0,C 180,E1 -985.253,E2 -985.253} C_VEL
LIN {X 0,Y 594.404,Z 571.439,A -85,B 0,C 180,E1 -987.968,E2 -987.968} C_VEL
LIN {X 0,Y 594.422,Z 571.443,A -85,B 0,C 180,E1 -990.678,E2 -990.678} C_VEL
LIN {X 0,Y 594.381,Z 571.44,A -85,B 0,C 180,E1 -993.39,E2 -993.39} C_VEL
LIN {X 0,Y 594.37,Z 571.443,A -85,B 0,C 180,E1 -996.11,E2 -996.11} C_VEL
LIN {X 0,Y 594.403,Z 571.445,A -85,B 0,C 180,E1 -998.843,E2 -998.843} C_VEL
LIN {X 0,Y 594.397,Z 571.438,A -85,B 0,C 180,E1 -1001.596,E2 -1001.596} C_VEL
LIN {X 0,Y 594.393,Z 571.442,A -85,B 0,C 180,E1 -1004.378,E2 -1004.378} C_VEL
LIN {X 0,Y 594.395,Z 571.443,A -85,B 0,C 180,E1 -1007.194,E2 -1007.194} C_VEL
LIN {X 0,Y 594.377,Z 571.44,A -85,B 0,C 180,E1 -1010.054,E2 -1010.054} C_VEL
LIN {X 0,Y 594.361,Z 571.454,A -85,B 0,C 180,E1 -1012.968,E2 -1012.968} C_VEL
LIN {X 0,Y 594.379,Z 571.448,A -85,B 0,C 180,E1 -1015.194,E2 -1015.194} C_VEL
LIN {X 0,Y 594.39,Z 571.442,A -85,B 0,C 180,E1 -1017.527,E2 -1017.527} C_VEL
LIN {X 0,Y 594.389,Z 571.439,A -85,B 0,C 180,E1 -1020.328,E2 -1020.328} C_VEL
LIN {X 0,Y 594.382,Z 571.447,A -85,B 0,C 180,E1 -1022.951,E2 -1022.951} C_VEL
LIN {X 0,Y 594.36,Z 571.449,A -85,B 0,C 180,E1 -1025.409,E2 -1025.409} C_VEL
LIN {X 0,Y 594.386,Z 571.44,A -85,B 0,C 180,E1 -1027.941,E2 -1027.941} C_VEL
LIN {X 0,Y 594.38,Z 571.443,A -85,B 0,C 180,E1 -1030.822,E2 -1030.822} C_VEL
LIN {X 0,Y 594.37,Z 571.452,A -85,B 0,C 180,E1 -1033.3,E2 -1033.3} C_VEL
LIN {X 0,Y 594.372,Z 571.441,A -85,B 0,C 180,E1 -1036.161,E2 -1036.161} C_VEL
LIN {X 0,Y 594.384,Z 571.439,A -85,B 0,C 180,E1 -1038.536,E2 -1038.536} C_VEL
LIN {X 0,Y 594.389,Z 571.446,A -85,B 0,C 180,E1 -1041.296,E2 -1041.296} C_VEL
LIN {X 0,Y 594.356,Z 571.45,A -85,B 0,C 180,E1 -1043.756,E2 -1043.756} C_VEL
LIN {X 0,Y 594.38,Z 571.441,A -85,B 0,C 180,E1 -1046.239,E2 -1046.239} C_VEL
LIN {X 0,Y 594.373,Z 571.44,A -85,B 0,C 180,E1 -1048.65,E2 -1048.65} C_VEL
LIN {X 0,Y 594.388,Z 571.44,A -85,B 0,C 180,E1 -1051.042,E2 -1051.042} C_VEL
LIN {X 0,Y 594.388,Z 571.445,A -85,B 0,C 180,E1 -1053.978,E2 -1053.978} C_VEL
LIN {X 0,Y 594.379,Z 571.442,A -85,B 0,C 180,E1 -1056.296,E2 -1056.296} C_VEL
LIN {X 0,Y 594.408,Z 571.438,A -85,B 0,C 180,E1 -1059.225,E2 -1059.225} C_VEL
LIN {X 0,Y 594.354,Z 571.45,A -85,B 0,C 180,E1 -1062.095,E2 -1062.095} C_VEL
LIN {X 0,Y 594.367,Z 571.447,A -85,B 0,C 180,E1 -1064.219,E2 -1064.219} C_VEL
LIN {X 0,Y 594.383,Z 571.444,A -85,B 0,C 180,E1 -1066.321,E2 -1066.321} C_VEL
LIN {X 0,Y 594.38,Z 571.44,A -85,B 0,C 180,E1 -1069.095,E2 -1069.095} C_VEL
LIN {X 0,Y 594.42,Z 571.442,A -85,B 0,C 180,E1 -1071.843,E2 -1071.843} C_VEL
LIN {X 0,Y 594.391,Z 571.441,A -85,B 0,C 180,E1 -1074.572,E2 -1074.572} C_VEL
LIN {X 0,Y 594.414,Z 571.436,A -85,B 0,C 180,E1 -1077.289,E2 -1077.289} C_VEL
LIN {X 0,Y 594.419,Z 571.442,A -85,B 0,C 180,E1 -1080,E2 -1080} C_VEL
LIN {X 0,Y 594.414,Z 571.439,A -85,B 0,C 180,E1 -1082.711,E2 -1082.711} C_VEL
LIN {X 0,Y 594.389,Z 571.439,A -85,B 0,C 180,E1 -1085.428,E2 -1085.428} C_VEL
LIN {X 0,Y 594.419,Z 571.443,A -85,B 0,C 180,E1 -1088.157,E2 -1088.157} C_VEL
LIN {X 0,Y 594.395,Z 571.439,A -85,B 0,C 180,E1 -1091.074,E2 -1091.074} C_VEL
LIN {X 0,Y 594.383,Z 571.44,A -85,B 0,C 180,E1 -1093.679,E2 -1093.679} C_VEL
LIN {X 0,Y 594.396,Z 571.445,A -85,B 0,C 180,E1 -1096.718,E2 -1096.718} C_VEL
LIN {X 0,Y 594.371,Z 571.441,A -85,B 0,C 180,E1 -1099.334,E2 -1099.334} C_VEL
LIN {X 0,Y 594.369,Z 571.441,A -85,B 0,C 180,E1 -1101.503,E2 -1101.503} C_VEL
LIN {X 0,Y 594.394,Z 571.445,A -85,B 0,C 180,E1 -1104.446,E2 -1104.446} C_VEL
LIN {X 0,Y 594.385,Z 571.45,A -85,B 0,C 180,E1 -1106.7,E2 -1106.7} C_VEL
LIN {X 0,Y 594.385,Z 571.445,A -85,B 0,C 180,E1 -1108.998,E2 -1108.998} C_VEL
LIN {X 0,Y 594.38,Z 571.44,A -85,B 0,C 180,E1 -1111.642,E2 -1111.642} C_VEL
LIN {X 0,Y 594.389,Z 571.445,A -85,B 0,C 180,E1 -1114.58,E2 -1114.58} C_VEL
LIN {X 0,Y 594.396,Z 571.439,A -85,B 0,C 180,E1 -1117.608,E2 -1117.608} C_VEL
LIN {X 0,Y 594.374,Z 571.445,A -85,B 0,C 180,E1 -1120.567,E2 -1120.567} C_VEL
LIN {X 0,Y 594.373,Z 571.446,A -85,B 0,C 180,E1 -1123.299,E2 -1123.299} C_VEL
LIN {X 0,Y 594.365,Z 571.442,A -85,B 0,C 180,E1 -1126.161,E2 -1126.161} C_VEL
LIN {X 0,Y 594.383,Z 571.442,A -85,B 0,C 180,E1 -1128.536,E2 -1128.536} C_VEL
LIN {X 0,Y 594.383,Z 571.447,A -85,B 0,C 180,E1 -1131.296,E2 -1131.296} C_VEL
LIN {X 0,Y 594.356,Z 571.445,A -85,B 0,C 180,E1 -1133.755,E2 -1133.755} C_VEL
LIN {X 0,Y 594.384,Z 571.439,A -85,B 0,C 180,E1 -1136.239,E2 -1136.239} C_VEL
LIN {X 0,Y 594.374,Z 571.442,A -85,B 0,C 180,E1 -1138.649,E2 -1138.649} C_VEL
LIN {X 0,Y 594.39,Z 571.445,A -85,B 0,C 180,E1 -1141.042,E2 -1141.042} C_VEL
LIN {X 0,Y 594.386,Z 571.442,A -85,B 0,C 180,E1 -1143.978,E2 -1143.978} C_VEL
LIN {X 0,Y 594.431,Z 571.597,A -85,B 0,C 180,E1 -1146.205,E2 -1146.205} C_VEL
LIN {X 0,Y 594.884,Z 575.009,A -85,B 0,C 180,E1 -1146.685,E2 -1146.685} C_VEL
LIN {X 0,Y 594.726,Z 596.845,A -85,B 0,C 180,E1 -1149.597,E2 -1149.597} C_VEL
LIN {X 0,Y 594.589,Z 620.046,A -85,B 0,C 180,E1 -1152.635,E2 -1152.635} C_VEL
LIN {X 0,Y 594.488,Z 643.246,A -85,B 0,C 180,E1 -1155.625,E2 -1155.625} C_VEL
LIN {X 0,Y 594.467,Z 651.349,A -85,B 0,C 180,E1 -1156.66,E2 -1156.66} C_VEL
LIN {X 0,Y 594.763,Z 657.453,A -85,B 0,C 180,E1 -1156.743,E2 -1156.743} C_VEL
LIN {X 0,Y 594.679,Z 759.911,A -85,B 0,C 180,E1 -1157.999,E2 -1157.999} C_VEL
LIN {X 0,Y 594.652,Z 772.434,A -85,B 0,C 180,E1 -1158.279,E2 -1158.279} C_VEL
LIN {X 0,Y 594.575,Z 785.256,A -85,B 0,C 180,E1 -1158.706,E2 -1158.706} C_VEL
LIN {X 0,Y 594.538,Z 797.62,A -85,B 0,C 180,E1 -1159.269,E2 -1159.269} C_VEL
LIN {X 0,Y 594.472,Z 809.189,A -85,B 0,C 180,E1 -1159.957,E2 -1159.957} C_VEL
LIN {X 0,Y 594.413,Z 819.587,A -85,B 0,C 180,E1 -1160.729,E2 -1160.729} C_VEL
LIN {X 0,Y 594.366,Z 828.105,A -85,B 0,C 180,E1 -1161.5,E2 -1161.5} C_VEL
LIN {X 0,Y 594.347,Z 835.955,A -85,B 0,C 180,E1 -1162.355,E2 -1162.355} C_VEL
LIN {X 0,Y 594.283,Z 843.81,A -85,B 0,C 180,E1 -1163.408,E2 -1163.408} C_VEL
LIN {X 0,Y 594.289,Z 850.677,A -85,B 0,C 180,E1 -1164.571,E2 -1164.571} C_VEL
LIN {X 0,Y 594.271,Z 855.368,A -85,B 0,C 180,E1 -1165.591,E2 -1165.591} C_VEL
LIN {X 0,Y 594.268,Z 858.954,A -85,B 0,C 180,E1 -1166.609,E2 -1166.609} C_VEL
LIN {X 0,Y 594.226,Z 860.807,A -85,B 0,C 180,E1 -1167.288,E2 -1167.288} C_VEL
LIN {X 0,Y 594.239,Z 862.2,A -85,B 0,C 180,E1 -1167.966,E2 -1167.966} C_VEL
LIN {X 0,Y 594.239,Z 863.783,A -85,B 0,C 180,E1 -1169.322,E2 -1169.322} C_VEL
LIN {X 0,Y 594.236,Z 864,A -85,B 0,C 180,E1 -1169.999,E2 -1169.999} C_VEL
LIN {X 0,Y 594.247,Z 863.185,A -85,B 0,C 180,E1 -1171.355,E2 -1171.355} C_VEL
LIN {X 0,Y 594.239,Z 862.203,A -85,B 0,C 180,E1 -1172.033,E2 -1172.033} C_VEL
LIN {X 0,Y 594.226,Z 860.811,A -85,B 0,C 180,E1 -1172.711,E2 -1172.711} C_VEL
LIN {X 0,Y 594.289,Z 857.898,A -85,B 0,C 180,E1 -1173.729,E2 -1173.729} C_VEL
LIN {X 0,Y 594.241,Z 853.953,A -85,B 0,C 180,E1 -1174.748,E2 -1174.748} C_VEL
LIN {X 0,Y 594.304,Z 847.882,A -85,B 0,C 180,E1 -1175.938,E2 -1175.938} C_VEL
LIN {X 0,Y 594.311,Z 841.242,A -85,B 0,C 180,E1 -1176.961,E2 -1176.961} C_VEL
LIN {X 0,Y 594.359,Z 832.996,A -85,B 0,C 180,E1 -1177.986,E2 -1177.986} C_VEL
LIN {X 0,Y 594.382,Z 824.546,A -85,B 0,C 180,E1 -1178.841,E2 -1178.841} C_VEL
LIN {X 0,Y 594.423,Z 814.104,A -85,B 0,C 180,E1 -1179.699,E2 -1179.699} C_VEL
LIN {X 0,Y 594.489,Z 803.771,A -85,B 0,C 180,E1 -1180.385,E2 -1180.385} C_VEL
LIN {X 0,Y 594.559,Z 792.708,A -85,B 0,C 180,E1 -1180.974,E2 -1180.974} C_VEL
LIN {X 0,Y 594.602,Z 780.726,A -85,B 0,C 180,E1 -1181.463,E2 -1181.463} C_VEL
LIN {X 0,Y 594.638,Z 767.386,A -85,B 0,C 180,E1 -1181.849,E2 -1181.849} C_VEL
LIN {X 0,Y 594.68,Z 754.146,A -85,B 0,C 180,E1 -1182.086,E2 -1182.086} C_VEL
LIN {X 0,Y 594.662,Z 652.882,A -85,B 0,C 180,E1 -1183.315,E2 -1183.315} C_VEL
LIN {X 0,Y 594.473,Z 651.276,A -85,B 0,C 180,E1 -1183.349,E2 -1183.349} C_VEL
LIN {X 0,Y 594.574,Z 626.881,A -85,B 0,C 180,E1 -1186.479,E2 -1186.479} C_VEL
LIN {X 0,Y 594.691,Z 603.681,A -85,B 0,C 180,E1 -1189.502,E2 -1189.502} C_VEL
LIN {X 0,Y 594.812,Z 580.914,A -85,B 0,C 180,E1 -1192.523,E2 -1192.523} C_VEL
LIN {X 0,Y 594.839,Z 573.656,A -85,B 0,C 180,E1 -1193.499,E2 -1193.499} C_VEL
LIN {X 0,Y 594.41,Z 571.443,A -85,B 0,C 180,E1 -1193.841,E2 -1193.841} C_VEL
LIN {X 0,Y 594.385,Z 571.449,A -85,B 0,C 180,E1 -1196.698,E2 -1196.698} C_VEL
LIN {X 0,Y 594.381,Z 571.444,A -85,B 0,C 180,E1 -1198.997,E2 -1198.997} C_VEL
LIN {X 0,Y 594.376,Z 571.441,A -85,B 0,C 180,E1 -1201.642,E2 -1201.642} C_VEL
LIN {X 0,Y 594.393,Z 571.449,A -85,B 0,C 180,E1 -1204.578,E2 -1204.578} C_VEL
LIN {X 0,Y 594.381,Z 571.442,A -85,B 0,C 180,E1 -1207.086,E2 -1207.086} C_VEL
LIN {X 0,Y 594.374,Z 571.442,A -85,B 0,C 180,E1 -1209.774,E2 -1209.774} C_VEL
LIN {X 0,Y 594.366,Z 571.451,A -85,B 0,C 180,E1 -1212.374,E2 -1212.374} C_VEL
LIN {X 0,Y 594.358,Z 571.444,A -85,B 0,C 180,E1 -1215.19,E2 -1215.19} C_VEL
LIN {X 0,Y 594.368,Z 571.442,A -85,B 0,C 180,E1 -1217.624,E2 -1217.624} C_VEL
LIN {X 0,Y 594.392,Z 571.447,A -85,B 0,C 180,E1 -1220.321,E2 -1220.321} C_VEL
LIN {X 0,Y 594.384,Z 571.443,A -85,B 0,C 180,E1 -1222.913,E2 -1222.913} C_VEL
LIN {X 0,Y 594.382,Z 571.442,A -85,B 0,C 180,E1 -1225.86,E2 -1225.86} C_VEL
LIN {X 0,Y 594.386,Z 571.446,A -85,B 0,C 180,E1 -1228.651,E2 -1228.651} C_VEL
LIN {X 0,Y 594.377,Z 571.442,A -85,B 0,C 180,E1 -1231.041,E2 -1231.041} C_VEL
LIN {X 0,Y 594.389,Z 571.442,A -85,B 0,C 180,E1 -1233.974,E2 -1233.974} C_VEL
LIN {X 0,Y 594.387,Z 571.448,A -85,B 0,C 180,E1 -1236.296,E2 -1236.296} C_VEL
LIN {X 0,Y 594.4,Z 571.438,A -85,B 0,C 180,E1 -1239.224,E2 -1239.224} C_VEL
LIN {X 0,Y 594.375,Z 571.447,A -85,B 0,C 180,E1 -1242.096,E2 -1242.096} C_VEL
LIN {X 0,Y 594.363,Z 571.45,A -85,B 0,C 180,E1 -1244.219,E2 -1244.219} C_VEL
LIN {X 0,Y 594.363,Z 571.444,A -85,B 0,C 180,E1 -1247.017,E2 -1247.017} C_VEL
LIN {X 0,Y 594.39,Z 571.441,A -85,B 0,C 180,E1 -1249.784,E2 -1249.784} C_VEL
LIN {X 0,Y 594.386,Z 571.447,A -85,B 0,C 180,E1 -1252.527,E2 -1252.527} C_VEL
LIN {X 0,Y 594.399,Z 571.438,A -85,B 0,C 180,E1 -1255.252,E2 -1255.252} C_VEL
LIN {X 0,Y 594.388,Z 571.444,A -85,B 0,C 180,E1 -1257.967,E2 -1257.967} C_VEL
LIN {X 0,Y 594.418,Z 571.44,A -85,B 0,C 180,E1 -1260.677,E2 -1260.677} C_VEL
LIN {X 0,Y 594.376,Z 571.441,A -85,B 0,C 180,E1 -1263.389,E2 -1263.389} C_VEL
LIN {X 0,Y 594.385,Z 571.448,A -85,B 0,C 180,E1 -1266.109,E2 -1266.109} C_VEL
LIN {X 0,Y 594.398,Z 571.44,A -85,B 0,C 180,E1 -1268.842,E2 -1268.842} C_VEL
LIN {X 0,Y 594.388,Z 571.441,A -85,B 0,C 180,E1 -1271.596,E2 -1271.596} C_VEL
LIN {X 0,Y 594.383,Z 571.45,A -85,B 0,C 180,E1 -1274.377,E2 -1274.377} C_VEL
LIN {X 0,Y 594.358,Z 571.444,A -85,B 0,C 180,E1 -1275.339,E2 -1275.339} C_VEL
LIN {X 0,Y 593.68,Z 571.532,A -85,B 0,C 180,E1 -1275.717,E2 -1275.717} C_VEL
LIN {X 0,Y 588.017,Z 572.238,A -85,B 0,C 180,E1 -1276.903,E2 -1276.903} C_VEL
LIN {X 0,Y 587.361,Z 572.317,A -85,B 0,C 180,E1 -1277.287,E2 -1277.287} C_VEL
LIN {X 0,Y 587.395,Z 572.508,A -85,B 0,C 180,E1 -1277.539,E2 -1277.539} C_VEL
LIN {X 0,Y 587.35,Z 585.187,A -85,B 0,C 180,E1 -1279.939,E2 -1279.939} C_VEL
LIN {X 0,Y 587.342,Z 593.863,A -85,B 0,C 180,E1 -1281.566,E2 -1281.566} C_VEL
LIN {X 0,Y 587.842,Z 598.274,A -85,B 0,C 180,E1 -1281.639,E2 -1281.639} C_VEL
LIN {X 0,Y 587.71,Z 700.626,A -85,B 0,C 180,E1 -1282.913,E2 -1282.913} C_VEL
LIN {X 0,Y 587.676,Z 714.112,A -85,B 0,C 180,E1 -1283.232,E2 -1283.232} C_VEL
LIN {X 0,Y 587.608,Z 726.573,A -85,B 0,C 180,E1 -1283.667,E2 -1283.667} C_VEL
LIN {X 0,Y 587.533,Z 738.918,A -85,B 0,C 180,E1 -1284.256,E2 -1284.256} C_VEL
LIN {X 0,Y 587.439,Z 750.125,A -85,B 0,C 180,E1 -1284.943,E2 -1284.943} C_VEL
LIN {X 0,Y 587.362,Z 761.236,A -85,B 0,C 180,E1 -1285.801,E2 -1285.801} C_VEL
LIN {X 0,Y 587.285,Z 770.255,A -85,B 0,C 180,E1 -1286.664,E2 -1286.664} C_VEL
LIN {X 0,Y 587.266,Z 778.899,A -85,B 0,C 180,E1 -1287.679,E2 -1287.679} C_VEL
LIN {X 0,Y 587.214,Z 785.305,A -85,B 0,C 180,E1 -1288.603,E2 -1288.603} C_VEL
LIN {X 0,Y 587.197,Z 791.842,A -85,B 0,C 180,E1 -1289.782,E2 -1289.782} C_VEL
LIN {X 0,Y 587.164,Z 796.859,A -85,B 0,C 180,E1 -1290.976,E2 -1290.976} C_VEL
LIN {X 0,Y 587.135,Z 799.531,A -85,B 0,C 180,E1 -1291.805,E2 -1291.805} C_VEL
LIN {X 0,Y 587.135,Z 802.356,A -85,B 0,C 180,E1 -1293.083,E2 -1293.083} C_VEL
LIN {X 0,Y 587.132,Z 803.756,A -85,B 0,C 180,E1 -1294.319,E2 -1294.319} C_VEL
LIN {X 0,Y 587.136,Z 803.899,A -85,B 0,C 180,E1 -1295.517,E2 -1295.517} C_VEL
LIN {X 0,Y 587.124,Z 802.745,A -85,B 0,C 180,E1 -1296.763,E2 -1296.763} C_VEL
LIN {X 0,Y 587.148,Z 800.725,A -85,B 0,C 180,E1 -1297.816,E2 -1297.816} C_VEL
LIN {X 0,Y 587.169,Z 797.538,A -85,B 0,C 180,E1 -1298.923,E2 -1298.923} C_VEL
LIN {X 0,Y 587.204,Z 793.254,A -85,B 0,C 180,E1 -1300.007,E2 -1300.007} C_VEL
LIN {X 0,Y 587.202,Z 787.227,A -85,B 0,C 180,E1 -1301.168,E2 -1301.168} C_VEL
LIN {X 0,Y 587.237,Z 779.635,A -85,B 0,C 180,E1 -1302.314,E2 -1302.314} C_VEL
LIN {X 0,Y 587.323,Z 771.567,A -85,B 0,C 180,E1 -1303.286,E2 -1303.286} C_VEL
LIN {X 0,Y 587.385,Z 761.421,A -85,B 0,C 180,E1 -1304.273,E2 -1304.273} C_VEL
LIN {X 0,Y 587.444,Z 750.769,A -85,B 0,C 180,E1 -1305.103,E2 -1305.103} C_VEL
LIN {X 0,Y 587.496,Z 740.173,A -85,B 0,C 180,E1 -1305.765,E2 -1305.765} C_VEL
LIN {X 0,Y 587.583,Z 728.595,A -85,B 0,C 180,E1 -1306.337,E2 -1306.337} C_VEL
LIN {X 0,Y 587.675,Z 715.851,A -85,B 0,C 180,E1 -1306.808,E2 -1306.808} C_VEL
LIN {X 0,Y 587.699,Z 702.519,A -85,B 0,C 180,E1 -1307.141,E2 -1307.141} C_VEL
LIN {X 0,Y 587.735,Z 681.135,A -85,B 0,C 180,E1 -1307.436,E2 -1307.436} C_VEL
LIN {X 0,Y 587.715,Z 596.379,A -85,B 0,C 180,E1 -1308.477,E2 -1308.477} C_VEL
LIN {X 0,Y 587.344,Z 593.823,A -85,B 0,C 180,E1 -1308.531,E2 -1308.531} C_VEL
LIN {X 0,Y 587.402,Z 577.891,A -85,B 0,C 180,E1 -1311.527,E2 -1311.527} C_VEL
LIN {X 0,Y 587.351,Z 572.319,A -85,B 0,C 180,E1 -1312.61,E2 -1312.61} C_VEL
LIN {X 0,Y 587.347,Z 572.317,A -85,B 0,C 180,E1 -1314.947,E2 -1314.947} C_VEL
LIN {X 0,Y 587.337,Z 572.32,A -85,B 0,C 180,E1 -1317.422,E2 -1317.422} C_VEL
LIN {X 0,Y 587.331,Z 572.326,A -85,B 0,C 180,E1 -1319.831,E2 -1319.831} C_VEL
LIN {X 0,Y 587.35,Z 572.322,A -85,B 0,C 180,E1 -1322.308,E2 -1322.308} C_VEL
LIN {X 0,Y 587.333,Z 572.322,A -85,B 0,C 180,E1 -1324.484,E2 -1324.484} C_VEL
LIN {X 0,Y 587.317,Z 572.32,A -85,B 0,C 180,E1 -1327.132,E2 -1327.132} C_VEL
LIN {X 0,Y 587.33,Z 572.321,A -85,B 0,C 180,E1 -1329.696,E2 -1329.696} C_VEL
LIN {X 0,Y 587.36,Z 572.319,A -85,B 0,C 180,E1 -1332.595,E2 -1332.595} C_VEL
LIN {X 0,Y 587.366,Z 572.316,A -85,B 0,C 180,E1 -1335.74,E2 -1335.74} C_VEL
LIN {X 0,Y 587.349,Z 572.318,A -85,B 0,C 180,E1 -1338.867,E2 -1338.867} C_VEL
LIN {X 0,Y 587.367,Z 572.315,A -85,B 0,C 180,E1 -1341.746,E2 -1341.746} C_VEL
LIN {X 0,Y 587.359,Z 572.324,A -85,B 0,C 180,E1 -1344.508,E2 -1344.508} C_VEL
LIN {X 0,Y 587.37,Z 572.314,A -85,B 0,C 180,E1 -1347.257,E2 -1347.257} C_VEL
LIN {X 0,Y 587.386,Z 572.313,A -85,B 0,C 180,E1 -1350.001,E2 -1350.001} C_VEL
LIN {X 0,Y 587.38,Z 572.32,A -85,B 0,C 180,E1 -1352.744,E2 -1352.744} C_VEL
LIN {X 0,Y 587.358,Z 572.315,A -85,B 0,C 180,E1 -1355.494,E2 -1355.494} C_VEL
LIN {X 0,Y 587.372,Z 572.316,A -85,B 0,C 180,E1 -1358.256,E2 -1358.256} C_VEL
LIN {X 0,Y 587.352,Z 572.32,A -85,B 0,C 180,E1 -1361.134,E2 -1361.134} C_VEL
LIN {X 0,Y 587.369,Z 572.315,A -85,B 0,C 180,E1 -1364.261,E2 -1364.261} C_VEL
LIN {X 0,Y 587.355,Z 572.317,A -85,B 0,C 180,E1 -1367.406,E2 -1367.406} C_VEL
LIN {X 0,Y 587.333,Z 572.319,A -85,B 0,C 180,E1 -1370.305,E2 -1370.305} C_VEL
LIN {X 0,Y 587.317,Z 572.325,A -85,B 0,C 180,E1 -1373.26,E2 -1373.26} C_VEL
LIN {X 0,Y 587.337,Z 572.32,A -85,B 0,C 180,E1 -1375.517,E2 -1375.517} C_VEL
LIN {X 0,Y 587.351,Z 572.316,A -85,B 0,C 180,E1 -1377.818,E2 -1377.818} C_VEL
LIN {X 0,Y 587.339,Z 572.319,A -85,B 0,C 180,E1 -1380.51,E2 -1380.51} C_VEL
LIN {X 0,Y 587.338,Z 572.324,A -85,B 0,C 180,E1 -1383.397,E2 -1383.397} C_VEL
LIN {X 0,Y 587.297,Z 572.323,A -85,B 0,C 180,E1 -1385.9,E2 -1385.9} C_VEL
LIN {X 0,Y 587.334,Z 572.318,A -85,B 0,C 180,E1 -1388.48,E2 -1388.48} C_VEL
LIN {X 0,Y 587.339,Z 572.325,A -85,B 0,C 180,E1 -1391.157,E2 -1391.157} C_VEL
LIN {X 0,Y 587.316,Z 572.32,A -85,B 0,C 180,E1 -1394.112,E2 -1394.112} C_VEL
LIN {X 0,Y 587.32,Z 572.323,A -85,B 0,C 180,E1 -1396.994,E2 -1396.994} C_VEL
LIN {X 0,Y 587.319,Z 572.325,A -85,B 0,C 180,E1 -1399.746,E2 -1399.746} C_VEL
LIN {X 0,Y 587.35,Z 572.316,A -85,B 0,C 180,E1 -1402.393,E2 -1402.393} C_VEL
LIN {X 0,Y 587.366,Z 572.32,A -85,B 0,C 180,E1 -1405.78,E2 -1405.78} C_VEL
LIN {X 0,Y 587.345,Z 572.318,A -85,B 0,C 180,E1 -1408.231,E2 -1408.231} C_VEL
LIN {X 0,Y 587.354,Z 572.315,A -85,B 0,C 180,E1 -1410.867,E2 -1410.867} C_VEL
LIN {X 0,Y 587.363,Z 572.323,A -85,B 0,C 180,E1 -1413.819,E2 -1413.819} C_VEL
LIN {X 0,Y 587.333,Z 572.324,A -85,B 0,C 180,E1 -1415.993,E2 -1415.993} C_VEL
LIN {X 0,Y 587.324,Z 572.322,A -85,B 0,C 180,E1 -1418.226,E2 -1418.226} C_VEL
LIN {X 0,Y 587.352,Z 572.316,A -85,B 0,C 180,E1 -1421.151,E2 -1421.151} C_VEL
LIN {X 0,Y 587.327,Z 572.327,A -85,B 0,C 180,E1 -1424.025,E2 -1424.025} C_VEL
LIN {X 0,Y 587.362,Z 572.321,A -85,B 0,C 180,E1 -1426.154,E2 -1426.154} C_VEL
LIN {X 0,Y 587.346,Z 572.316,A -85,B 0,C 180,E1 -1428.963,E2 -1428.963} C_VEL
LIN {X 0,Y 587.371,Z 572.318,A -85,B 0,C 180,E1 -1431.745,E2 -1431.745} C_VEL
LIN {X 0,Y 587.357,Z 572.318,A -85,B 0,C 180,E1 -1434.507,E2 -1434.507} C_VEL
LIN {X 0,Y 587.38,Z 572.312,A -85,B 0,C 180,E1 -1437.257,E2 -1437.257} C_VEL
LIN {X 0,Y 587.388,Z 572.318,A -85,B 0,C 180,E1 -1440,E2 -1440} C_VEL
LIN {X 0,Y 587.38,Z 572.315,A -85,B 0,C 180,E1 -1442.743,E2 -1442.743} C_VEL
LIN {X 0,Y 587.355,Z 572.315,A -85,B 0,C 180,E1 -1445.493,E2 -1445.493} C_VEL
LIN {X 0,Y 587.371,Z 572.322,A -85,B 0,C 180,E1 -1448.255,E2 -1448.255} C_VEL
LIN {X 0,Y 587.354,Z 572.316,A -85,B 0,C 180,E1 -1451.134,E2 -1451.134} C_VEL
LIN {X 0,Y 587.371,Z 572.32,A -85,B 0,C 180,E1 -1454.26,E2 -1454.26} C_VEL
LIN {X 0,Y 587.35,Z 572.315,A -85,B 0,C 180,E1 -1457.406,E2 -1457.406} C_VEL
LIN {X 0,Y 587.318,Z 572.319,A -85,B 0,C 180,E1 -1459.576,E2 -1459.576} C_VEL
LIN {X 0,Y 587.343,Z 572.326,A -85,B 0,C 180,E1 -1462.514,E2 -1462.514} C_VEL
LIN {X 0,Y 587.335,Z 572.318,A -85,B 0,C 180,E1 -1465.517,E2 -1465.517} C_VEL
LIN {X 0,Y 587.345,Z 572.316,A -85,B 0,C 180,E1 -1467.818,E2 -1467.818} C_VEL
LIN {X 0,Y 587.341,Z 572.323,A -85,B 0,C 180,E1 -1470.51,E2 -1470.51} C_VEL
LIN {X 0,Y 587.338,Z 572.319,A -85,B 0,C 180,E1 -1473.397,E2 -1473.397} C_VEL
LIN {X 0,Y 587.296,Z 572.322,A -85,B 0,C 180,E1 -1475.9,E2 -1475.9} C_VEL
LIN {X 0,Y 587.336,Z 572.321,A -85,B 0,C 180,E1 -1478.479,E2 -1478.479} C_VEL
LIN {X 0,Y 587.341,Z 572.324,A -85,B 0,C 180,E1 -1481.157,E2 -1481.157} C_VEL
LIN {X 0,Y 587.332,Z 572.318,A -85,B 0,C 180,E1 -1484.113,E2 -1484.113} C_VEL
LIN {X 0,Y 587.319,Z 572.33,A -85,B 0,C 180,E1 -1486.993,E2 -1486.993} C_VEL
LIN {X 0,Y 587.321,Z 572.32,A -85,B 0,C 180,E1 -1489.746,E2 -1489.746} C_VEL
LIN {X 0,Y 587.347,Z 572.316,A -85,B 0,C 180,E1 -1492.392,E2 -1492.392} C_VEL
LIN {X 0,Y 587.372,Z 572.315,A -85,B 0,C 180,E1 -1495.78,E2 -1495.78} C_VEL
LIN {X 0,Y 587.345,Z 572.316,A -85,B 0,C 180,E1 -1498.231,E2 -1498.231} C_VEL
LIN {X 0,Y 587.355,Z 572.319,A -85,B 0,C 180,E1 -1500.866,E2 -1500.866} C_VEL
LIN {X 0,Y 587.344,Z 572.321,A -85,B 0,C 180,E1 -1503.823,E2 -1503.823} C_VEL
LIN {X 0,Y 587.403,Z 572.45,A -85,B 0,C 180,E1 -1506.019,E2 -1506.019} C_VEL
LIN {X 0,Y 588,Z 576.374,A -85,B 0,C 180,E1 -1506.583,E2 -1506.583} C_VEL
LIN {X 0,Y 587.775,Z 599.575,A -85,B 0,C 180,E1 -1509.711,E2 -1509.711} C_VEL
LIN {X 0,Y 587.637,Z 622.616,A -85,B 0,C 180,E1 -1512.761,E2 -1512.761} C_VEL
LIN {X 0,Y 587.472,Z 646.221,A -85,B 0,C 180,E1 -1515.835,E2 -1515.835} C_VEL
LIN {X 0,Y 587.422,Z 651.349,A -85,B 0,C 180,E1 -1516.497,E2 -1516.497} C_VEL
LIN {X 0,Y 587.871,Z 655.664,A -85,B 0,C 180,E1 -1516.562,E2 -1516.562} C_VEL
LIN {X 0,Y 587.737,Z 759.911,A -85,B 0,C 180,E1 -1517.855,E2 -1517.855} C_VEL
LIN {X 0,Y 587.703,Z 772.435,A -85,B 0,C 180,E1 -1518.138,E2 -1518.138} C_VEL
LIN {X 0,Y 587.621,Z 785.019,A -85,B 0,C 180,E1 -1518.561,E2 -1518.561} C_VEL
LIN {X 0,Y 587.539,Z 797.619,A -85,B 0,C 180,E1 -1519.14,E2 -1519.14} C_VEL
LIN {X 0,Y 587.462,Z 809.19,A -85,B 0,C 180,E1 -1519.836,E2 -1519.836} C_VEL
LIN {X 0,Y 587.391,Z 819.588,A -85,B 0,C 180,E1 -1520.617,E2 -1520.617} C_VEL
LIN {X 0,Y 587.31,Z 828.105,A -85,B 0,C 180,E1 -1521.397,E2 -1521.397} C_VEL
LIN {X 0,Y 587.274,Z 835.955,A -85,B 0,C 180,E1 -1522.262,E2 -1522.262} C_VEL
LIN {X 0,Y 587.231,Z 842.465,A -85,B 0,C 180,E1 -1523.126,E2 -1523.126} C_VEL
LIN {X 0,Y 587.236,Z 848.862,A -85,B 0,C 180,E1 -1524.161,E2 -1524.161} C_VEL
LIN {X 0,Y 587.147,Z 853.947,A -85,B 0,C 180,E1 -1525.193,E2 -1525.193} C_VEL
LIN {X 0,Y 587.213,Z 857.893,A -85,B 0,C 180,E1 -1526.225,E2 -1526.225} C_VEL
LIN {X 0,Y 587.132,Z 860.807,A -85,B 0,C 180,E1 -1527.255,E2 -1527.255} C_VEL
LIN {X 0,Y 587.138,Z 862.2,A -85,B 0,C 180,E1 -1527.941,E2 -1527.941} C_VEL
LIN {X 0,Y 587.14,Z 863.784,A -85,B 0,C 180,E1 -1529.313,E2 -1529.313} C_VEL
LIN {X 0,Y 587.137,Z 864,A -85,B 0,C 180,E1 -1529.999,E2 -1529.999} C_VEL
LIN {X 0,Y 587.147,Z 863.186,A -85,B 0,C 180,E1 -1531.371,E2 -1531.371} C_VEL
LIN {X 0,Y 587.138,Z 862.203,A -85,B 0,C 180,E1 -1532.057,E2 -1532.057} C_VEL
LIN {X 0,Y 587.132,Z 860.811,A -85,B 0,C 180,E1 -1532.744,E2 -1532.744} C_VEL
LIN {X 0,Y 587.213,Z 857.898,A -85,B 0,C 180,E1 -1533.774,E2 -1533.774} C_VEL
LIN {X 0,Y 587.147,Z 853.953,A -85,B 0,C 180,E1 -1534.806,E2 -1534.806} C_VEL
LIN {X 0,Y 587.217,Z 847.882,A -85,B 0,C 180,E1 -1536.01,E2 -1536.01} C_VEL
LIN {X 0,Y 587.246,Z 841.242,A -85,B 0,C 180,E1 -1537.045,E2 -1537.045} C_VEL
LIN {X 0,Y 587.299,Z 832.997,A -85,B 0,C 180,E1 -1538.082,E2 -1538.082} C_VEL
LIN {X 0,Y 587.343,Z 824.546,A -85,B 0,C 180,E1 -1538.948,E2 -1538.948} C_VEL
LIN {X 0,Y 587.411,Z 814.105,A -85,B 0,C 180,E1 -1539.816,E2 -1539.816} C_VEL
LIN {X 0,Y 587.506,Z 803.772,A -85,B 0,C 180,E1 -1540.51,E2 -1540.51} C_VEL
LIN {X 0,Y 587.582,Z 791.818,A -85,B 0,C 180,E1 -1541.148,E2 -1541.148} C_VEL
LIN {X 0,Y 587.629,Z 779.615,A -85,B 0,C 180,E1 -1541.639,E2 -1541.639} C_VEL
LIN {X 0,Y 587.677,Z 766.471,A -85,B 0,C 180,E1 -1542.014,E2 -1542.014} C_VEL
LIN {X 0,Y 587.763,Z 754.146,A -85,B 0,C 180,E1 -1542.231,E2 -1542.231} C_VEL
LIN {X 0,Y 587.745,Z 653.553,A -85,B 0,C 180,E1 -1543.467,E2 -1543.467} C_VEL
LIN {X 0,Y 587.426,Z 651.276,A -85,B 0,C 180,E1 -1543.513,E2 -1543.513} C_VEL
LIN {X 0,Y 587.569,Z 629.611,A -85,B 0,C 180,E1 -1546.324,E2 -1546.324} C_VEL
LIN {X 0,Y 587.734,Z 607.102,A -85,B 0,C 180,E1 -1549.287,E2 -1549.287} C_VEL
LIN {X 0,Y 587.859,Z 585.939,A -85,B 0,C 180,E1 -1552.122,E2 -1552.122} C_VEL
LIN {X 0,Y 587.899,Z 575.021,A -85,B 0,C 180,E1 -1553.607,E2 -1553.607} C_VEL
LIN {X 0,Y 587.359,Z 572.323,A -85,B 0,C 180,E1 -1554.005,E2 -1554.005} C_VEL
LIN {X 0,Y 587.329,Z 572.323,A -85,B 0,C 180,E1 -1557.045,E2 -1557.045} C_VEL
LIN {X 0,Y 587.346,Z 572.318,A -85,B 0,C 180,E1 -1559.379,E2 -1559.379} C_VEL
LIN {X 0,Y 587.343,Z 572.319,A -85,B 0,C 180,E1 -1561.835,E2 -1561.835} C_VEL
LIN {X 0,Y 587.353,Z 572.323,A -85,B 0,C 180,E1 -1564.348,E2 -1564.348} C_VEL
LIN {X 0,Y 587.35,Z 572.323,A -85,B 0,C 180,E1 -1566.746,E2 -1566.746} C_VEL
LIN {X 0,Y 587.343,Z 572.318,A -85,B 0,C 180,E1 -1569.358,E2 -1569.358} C_VEL
LIN {X 0,Y 587.331,Z 572.323,A -85,B 0,C 180,E1 -1572.107,E2 -1572.107} C_VEL
LIN {X 0,Y 587.311,Z 572.323,A -85,B 0,C 180,E1 -1575.088,E2 -1575.088} C_VEL
LIN {X 0,Y 587.348,Z 572.319,A -85,B 0,C 180,E1 -1577.927,E2 -1577.927} C_VEL
LIN {X 0,Y 587.332,Z 572.32,A -85,B 0,C 180,E1 -1581.057,E2 -1581.057} C_VEL
LIN {X 0,Y 587.349,Z 572.316,A -85,B 0,C 180,E1 -1583.291,E2 -1583.291} C_VEL
LIN {X 0,Y 587.363,Z 572.316,A -85,B 0,C 180,E1 -1585.78,E2 -1585.78} C_VEL
LIN {X 0,Y 587.348,Z 572.323,A -85,B 0,C 180,E1 -1588.231,E2 -1588.231} C_VEL
LIN {X 0,Y 587.345,Z 572.32,A -85,B 0,C 180,E1 -1590.865,E2 -1590.865} C_VEL
LIN {X 0,Y 587.357,Z 572.317,A -85,B 0,C 180,E1 -1593.817,E2 -1593.817} C_VEL
LIN {X 0,Y 587.332,Z 572.322,A -85,B 0,C 180,E1 -1595.993,E2 -1595.993} C_VEL
LIN {X 0,Y 587.316,Z 572.328,A -85,B 0,C 180,E1 -1598.225,E2 -1598.225} C_VEL
LIN {X 0,Y 587.344,Z 572.317,A -85,B 0,C 180,E1 -1601.151,E2 -1601.151} C_VEL
LIN {X 0,Y 587.343,Z 572.317,A -85,B 0,C 180,E1 -1603.311,E2 -1603.311} C_VEL
LIN {X 0,Y 587.352,Z 572.322,A -85,B 0,C 180,E1 -1606.154,E2 -1606.154} C_VEL
LIN {X 0,Y 587.338,Z 572.319,A -85,B 0,C 180,E1 -1608.962,E2 -1608.962} C_VEL
LIN {X 0,Y 587.366,Z 572.316,A -85,B 0,C 180,E1 -1611.745,E2 -1611.745} C_VEL
LIN {X 0,Y 587.35,Z 572.324,A -85,B 0,C 180,E1 -1614.507,E2 -1614.507} C_VEL
LIN {X 0,Y 587.376,Z 572.313,A -85,B 0,C 180,E1 -1617.257,E2 -1617.257} C_VEL
LIN {X 0,Y 587.375,Z 572.318,A -85,B 0,C 180,E1 -1620,E2 -1620} C_VEL
LIN {X 0,Y 587.376,Z 572.317,A -85,B 0,C 180,E1 -1622.743,E2 -1622.743} C_VEL
LIN {X 0,Y 587.357,Z 572.316,A -85,B 0,C 180,E1 -1625.493,E2 -1625.493} C_VEL
LIN {X 0,Y 587.367,Z 572.325,A -85,B 0,C 180,E1 -1628.255,E2 -1628.255} C_VEL
LIN {X 0,Y 587.354,Z 572.316,A -85,B 0,C 180,E1 -1631.141,E2 -1631.141} C_VEL
LIN {X 0,Y 587.357,Z 572.327,A -85,B 0,C 180,E1 -1634.261,E2 -1634.261} C_VEL
LIN {X 0,Y 587.361,Z 572.317,A -85,B 0,C 180,E1 -1637.287,E2 -1637.287} C_VEL
LIN {X 0,Y 587.129,Z 573.075,A -85,B 0,C 180,E1 -1637.621,E2 -1637.621} C_VEL
LIN {X 0,Y 586.271,Z 575.192,A -85,B 0,C 180,E1 -1638.017,E2 -1638.017} C_VEL
LIN {X 0,Y 581.024,Z 583.691,A -85,B 0,C 180,E1 -1639.467,E2 -1639.467} C_VEL
LIN {X 0,Y 580.315,Z 586.368,A -85,B 0,C 180,E1 -1639.977,E2 -1639.977} C_VEL
LIN {X 0,Y 580.291,Z 593.956,A -85,B 0,C 180,E1 -1641.407,E2 -1641.407} C_VEL
LIN {X 0,Y 580.961,Z 598.652,A -85,B 0,C 180,E1 -1641.482,E2 -1641.482} C_VEL
LIN {X 0,Y 580.778,Z 700.268,A -85,B 0,C 180,E1 -1642.759,E2 -1642.759} C_VEL
LIN {X 0,Y 580.722,Z 713.519,A -85,B 0,C 180,E1 -1643.071,E2 -1643.071} C_VEL
LIN {X 0,Y 580.676,Z 725.21,A -85,B 0,C 180,E1 -1643.475,E2 -1643.475} C_VEL
LIN {X 0,Y 580.552,Z 737.002,A -85,B 0,C 180,E1 -1644.02,E2 -1644.02} C_VEL
LIN {X 0,Y 580.47,Z 748.144,A -85,B 0,C 180,E1 -1644.684,E2 -1644.684} C_VEL
LIN {X 0,Y 580.361,Z 758.556,A -85,B 0,C 180,E1 -1645.461,E2 -1645.461} C_VEL
LIN {X 0,Y 580.299,Z 768.118,A -85,B 0,C 180,E1 -1646.338,E2 -1646.338} C_VEL
LIN {X 0,Y 580.21,Z 775.929,A -85,B 0,C 180,E1 -1647.21,E2 -1647.21} C_VEL
LIN {X 0,Y 580.178,Z 783.173,A -85,B 0,C 180,E1 -1648.192,E2 -1648.192} C_VEL
LIN {X 0,Y 580.142,Z 789.65,A -85,B 0,C 180,E1 -1649.284,E2 -1649.284} C_VEL
LIN {X 0,Y 580.095,Z 795.606,A -85,B 0,C 180,E1 -1650.587,E2 -1650.587} C_VEL
LIN {X 0,Y 580.069,Z 798.432,A -85,B 0,C 180,E1 -1651.398,E2 -1651.398} C_VEL
LIN {X 0,Y 580.038,Z 800.681,A -85,B 0,C 180,E1 -1652.217,E2 -1652.217} C_VEL
LIN {X 0,Y 580.054,Z 802.706,A -85,B 0,C 180,E1 -1653.281,E2 -1653.281} C_VEL
LIN {X 0,Y 580.045,Z 803.888,A -85,B 0,C 180,E1 -1654.524,E2 -1654.524} C_VEL
LIN {X 0,Y 580.032,Z 803.791,A -85,B 0,C 180,E1 -1655.729,E2 -1655.729} C_VEL
LIN {X 0,Y 580.032,Z 802.561,A -85,B 0,C 180,E1 -1656.901,E2 -1656.901} C_VEL
LIN {X 0,Y 580.065,Z 799.946,A -85,B 0,C 180,E1 -1658.164,E2 -1658.164} C_VEL
LIN {X 0,Y 580.081,Z 795.504,A -85,B 0,C 180,E1 -1659.529,E2 -1659.529} C_VEL
LIN {X 0,Y 580.109,Z 791.068,A -85,B 0,C 180,E1 -1660.531,E2 -1660.531} C_VEL
LIN {X 0,Y 580.125,Z 785.568,A -85,B 0,C 180,E1 -1661.523,E2 -1661.523} C_VEL
LIN {X 0,Y 580.178,Z 778.821,A -85,B 0,C 180,E1 -1662.512,E2 -1662.512} C_VEL
LIN {X 0,Y 580.267,Z 770.55,A -85,B 0,C 180,E1 -1663.496,E2 -1663.496} C_VEL
LIN {X 0,Y 580.355,Z 761.247,A -85,B 0,C 180,E1 -1664.401,E2 -1664.401} C_VEL
LIN {X 0,Y 580.458,Z 750.48,A -85,B 0,C 180,E1 -1665.245,E2 -1665.245} C_VEL
LIN {X 0,Y 580.52,Z 739.85,A -85,B 0,C 180,E1 -1665.914,E2 -1665.914} C_VEL
LIN {X 0,Y 580.633,Z 727.89,A -85,B 0,C 180,E1 -1666.505,E2 -1666.505} C_VEL
LIN {X 0,Y 580.734,Z 714.819,A -85,B 0,C 180,E1 -1666.982,E2 -1666.982} C_VEL
LIN {X 0,Y 580.755,Z 701.445,A -85,B 0,C 180,E1 -1667.309,E2 -1667.309} C_VEL
LIN {X 0,Y 580.872,Z 667.022,A -85,B 0,C 180,E1 -1667.76,E2 -1667.76} C_VEL
LIN {X 0,Y 580.888,Z 597.645,A -85,B 0,C 180,E1 -1668.623,E2 -1668.623} C_VEL
LIN {X 0,Y 580.279,Z 593.852,A -85,B 0,C 180,E1 -1668.693,E2 -1668.693} C_VEL
LIN {X 0,Y 580.391,Z 578.362,A -85,B 0,C 180,E1 -1671.642,E2 -1671.642} C_VEL
LIN {X 0,Y 580.323,Z 573.195,A -85,B 0,C 180,E1 -1672.68,E2 -1672.68} C_VEL
LIN {X 0,Y 580.302,Z 573.198,A -85,B 0,C 180,E1 -1675.441,E2 -1675.441} C_VEL
LIN {X 0,Y 580.301,Z 573.205,A -85,B 0,C 180,E1 -1677.97,E2 -1677.97} C_VEL
LIN {X 0,Y 580.3,Z 573.195,A -85,B 0,C 180,E1 -1680.691,E2 -1680.691} C_VEL
LIN {X 0,Y 580.275,Z 573.198,A -85,B 0,C 180,E1 -1683.378,E2 -1683.378} C_VEL
LIN {X 0,Y 580.3,Z 573.198,A -85,B 0,C 180,E1 -1685.685,E2 -1685.685} C_VEL
LIN {X 0,Y 580.274,Z 573.204,A -85,B 0,C 180,E1 -1687.948,E2 -1687.948} C_VEL
LIN {X 0,Y 580.299,Z 573.195,A -85,B 0,C 180,E1 -1690.914,E2 -1690.914} C_VEL
LIN {X 0,Y 580.312,Z 573.192,A -85,B 0,C 180,E1 -1693.104,E2 -1693.104} C_VEL
LIN {X 0,Y 580.328,Z 573.196,A -85,B 0,C 180,E1 -1695.984,E2 -1695.984} C_VEL
LIN {X 0,Y 580.305,Z 573.196,A -85,B 0,C 180,E1 -1698.828,E2 -1698.828} C_VEL
LIN {X 0,Y 580.33,Z 573.191,A -85,B 0,C 180,E1 -1701.645,E2 -1701.645} C_VEL
LIN {X 0,Y 580.325,Z 573.202,A -85,B 0,C 180,E1 -1704.441,E2 -1704.441} C_VEL
LIN {X 0,Y 580.337,Z 573.19,A -85,B 0,C 180,E1 -1707.224,E2 -1707.224} C_VEL
LIN {X 0,Y 580.355,Z 573.189,A -85,B 0,C 180,E1 -1710.001,E2 -1710.001} C_VEL
LIN {X 0,Y 580.346,Z 573.196,A -85,B 0,C 180,E1 -1712.777,E2 -1712.777} C_VEL
LIN {X 0,Y 580.324,Z 573.191,A -85,B 0,C 180,E1 -1715.56,E2 -1715.56} C_VEL
LIN {X 0,Y 580.337,Z 573.194,A -85,B 0,C 180,E1 -1718.357,E2 -1718.357} C_VEL
LIN {X 0,Y 580.303,Z 573.197,A -85,B 0,C 180,E1 -1721.192,E2 -1721.192} C_VEL
LIN {X 0,Y 580.33,Z 573.19,A -85,B 0,C 180,E1 -1724.018,E2 -1724.018} C_VEL
LIN {X 0,Y 580.316,Z 573.202,A -85,B 0,C 180,E1 -1726.914,E2 -1726.914} C_VEL
LIN {X 0,Y 580.292,Z 573.195,A -85,B 0,C 180,E1 -1729.823,E2 -1729.823} C_VEL
LIN {X 0,Y 580.276,Z 573.197,A -85,B 0,C 180,E1 -1732.053,E2 -1732.053} C_VEL
LIN {X 0,Y 580.31,Z 573.202,A -85,B 0,C 180,E1 -1735.08,E2 -1735.08} C_VEL
LIN {X 0,Y 580.304,Z 573.193,A -85,B 0,C 180,E1 -1738.186,E2 -1738.186} C_VEL
LIN {X 0,Y 580.287,Z 573.199,A -85,B 0,C 180,E1 -1740.695,E2 -1740.695} C_VEL
LIN {X 0,Y 580.307,Z 573.201,A -85,B 0,C 180,E1 -1743.317,E2 -1743.317} C_VEL
LIN {X 0,Y 580.253,Z 573.202,A -85,B 0,C 180,E1 -1745.757,E2 -1745.757} C_VEL
LIN {X 0,Y 580.292,Z 573.195,A -85,B 0,C 180,E1 -1748.147,E2 -1748.147} C_VEL
LIN {X 0,Y 580.303,Z 573.197,A -85,B 0,C 180,E1 -1750.844,E2 -1750.844} C_VEL
LIN {X 0,Y 580.277,Z 573.202,A -85,B 0,C 180,E1 -1753.659,E2 -1753.659} C_VEL
LIN {X 0,Y 580.282,Z 573.196,A -85,B 0,C 180,E1 -1756.61,E2 -1756.61} C_VEL
LIN {X 0,Y 580.303,Z 573.199,A -85,B 0,C 180,E1 -1759.157,E2 -1759.157} C_VEL
LIN {X 0,Y 580.295,Z 573.198,A -85,B 0,C 180,E1 -1761.927,E2 -1761.927} C_VEL
LIN {X 0,Y 580.255,Z 573.199,A -85,B 0,C 180,E1 -1764.453,E2 -1764.453} C_VEL
LIN {X 0,Y 580.295,Z 573.196,A -85,B 0,C 180,E1 -1766.975,E2 -1766.975} C_VEL
LIN {X 0,Y 580.3,Z 573.201,A -85,B 0,C 180,E1 -1769.425,E2 -1769.425} C_VEL
LIN {X 0,Y 580.303,Z 573.197,A -85,B 0,C 180,E1 -1772.142,E2 -1772.142} C_VEL
LIN {X 0,Y 580.326,Z 573.194,A -85,B 0,C 180,E1 -1775.27,E2 -1775.27} C_VEL
LIN {X 0,Y 580.276,Z 573.205,A -85,B 0,C 180,E1 -1777.948,E2 -1777.948} C_VEL
LIN {X 0,Y 580.302,Z 573.193,A -85,B 0,C 180,E1 -1780.914,E2 -1780.914} C_VEL
LIN {X 0,Y 580.282,Z 573.206,A -85,B 0,C 180,E1 -1783.826,E2 -1783.826} C_VEL
LIN {X 0,Y 580.329,Z 573.2,A -85,B 0,C 180,E1 -1785.983,E2 -1785.983} C_VEL
LIN {X 0,Y 580.31,Z 573.193,A -85,B 0,C 180,E1 -1788.827,E2 -1788.827} C_VEL
LIN {X 0,Y 580.334,Z 573.194,A -85,B 0,C 180,E1 -1791.644,E2 -1791.644} C_VEL
LIN {X 0,Y 580.324,Z 573.195,A -85,B 0,C 180,E1 -1794.44,E2 -1794.44} C_VEL
LIN {X 0,Y 580.345,Z 573.188,A -85,B 0,C 180,E1 -1797.224,E2 -1797.224} C_VEL
LIN {X 0,Y 580.358,Z 573.194,A -85,B 0,C 180,E1 -1800,E2 -1800} C_VEL
LIN {X 0,Y 580.346,Z 573.19,A -85,B 0,C 180,E1 -1802.777,E2 -1802.777} C_VEL
LIN {X 0,Y 580.321,Z 573.192,A -85,B 0,C 180,E1 -1805.56,E2 -1805.56} C_VEL
LIN {X 0,Y 580.334,Z 573.201,A -85,B 0,C 180,E1 -1808.356,E2 -1808.356} C_VEL
LIN {X 0,Y 580.306,Z 573.193,A -85,B 0,C 180,E1 -1811.191,E2 -1811.191} C_VEL
LIN {X 0,Y 580.33,Z 573.194,A -85,B 0,C 180,E1 -1814.017,E2 -1814.017} C_VEL
LIN {X 0,Y 580.318,Z 573.195,A -85,B 0,C 180,E1 -1816.914,E2 -1816.914} C_VEL
LIN {X 0,Y 580.293,Z 573.195,A -85,B 0,C 180,E1 -1819.823,E2 -1819.823} C_VEL
LIN {X 0,Y 580.276,Z 573.199,A -85,B 0,C 180,E1 -1822.053,E2 -1822.053} C_VEL
LIN {X 0,Y 580.31,Z 573.196,A -85,B 0,C 180,E1 -1825.08,E2 -1825.08} C_VEL
LIN {X 0,Y 580.301,Z 573.196,A -85,B 0,C 180,E1 -1828.186,E2 -1828.186} C_VEL
LIN {X 0,Y 580.289,Z 573.205,A -85,B 0,C 180,E1 -1830.694,E2 -1830.694} C_VEL
LIN {X 0,Y 580.307,Z 573.195,A -85,B 0,C 180,E1 -1833.316,E2 -1833.316} C_VEL
LIN {X 0,Y 580.251,Z 573.2,A -85,B 0,C 180,E1 -1835.756,E2 -1835.756} C_VEL
LIN {X 0,Y 580.294,Z 573.195,A -85,B 0,C 180,E1 -1838.146,E2 -1838.146} C_VEL
LIN {X 0,Y 580.303,Z 573.203,A -85,B 0,C 180,E1 -1840.843,E2 -1840.843} C_VEL
LIN {X 0,Y 580.285,Z 573.197,A -85,B 0,C 180,E1 -1843.658,E2 -1843.658} C_VEL
LIN {X 0,Y 580.279,Z 573.2,A -85,B 0,C 180,E1 -1846.609,E2 -1846.609} C_VEL
LIN {X 0,Y 580.303,Z 573.203,A -85,B 0,C 180,E1 -1849.156,E2 -1849.156} C_VEL
LIN {X 0,Y 580.293,Z 573.195,A -85,B 0,C 180,E1 -1851.927,E2 -1851.927} C_VEL
LIN {X 0,Y 580.263,Z 573.199,A -85,B 0,C 180,E1 -1854.453,E2 -1854.453} C_VEL
LIN {X 0,Y 580.297,Z 573.201,A -85,B 0,C 180,E1 -1856.975,E2 -1856.975} C_VEL
LIN {X 0,Y 580.292,Z 573.204,A -85,B 0,C 180,E1 -1859.424,E2 -1859.424} C_VEL
LIN {X 0,Y 580.298,Z 573.195,A -85,B 0,C 180,E1 -1862.142,E2 -1862.142} C_VEL
LIN {X 0,Y 580.326,Z 573.201,A -85,B 0,C 180,E1 -1865.269,E2 -1865.269} C_VEL
LIN {X 0,Y 580.343,Z 573.303,A -85,B 0,C 180,E1 -1865.828,E2 -1865.828} C_VEL
LIN {X 0,Y 581.111,Z 577.739,A -85,B 0,C 180,E1 -1866.477,E2 -1866.477} C_VEL
LIN {X 0,Y 580.861,Z 599.575,A -85,B 0,C 180,E1 -1869.458,E2 -1869.458} C_VEL
LIN {X 0,Y 580.674,Z 620.046,A -85,B 0,C 180,E1 -1872.205,E2 -1872.205} C_VEL
LIN {X 0,Y 580.487,Z 641.882,A -85,B 0,C 180,E1 -1875.091,E2 -1875.091} C_VEL
LIN {X 0,Y 580.435,Z 651.349,A -85,B 0,C 180,E1 -1876.331,E2 -1876.331} C_VEL
LIN {X 0,Y 580.973,Z 657.453,A -85,B 0,C 180,E1 -1876.422,E2 -1876.422} C_VEL
LIN {X 0,Y 580.819,Z 759.911,A -85,B 0,C 180,E1 -1877.708,E2 -1877.708} C_VEL
LIN {X 0,Y 580.751,Z 772.434,A -85,B 0,C 180,E1 -1877.994,E2 -1877.994} C_VEL
LIN {X 0,Y 580.657,Z 785.354,A -85,B 0,C 180,E1 -1878.435,E2 -1878.435} C_VEL
LIN {X 0,Y 580.551,Z 797.618,A -85,B 0,C 180,E1 -1879.008,E2 -1879.008} C_VEL
LIN {X 0,Y 580.431,Z 809.192,A -85,B 0,C 180,E1 -1879.711,E2 -1879.711} C_VEL
LIN {X 0,Y 580.341,Z 819.589,A -85,B 0,C 180,E1 -1880.502,E2 -1880.502} C_VEL
LIN {X 0,Y 580.267,Z 828.105,A -85,B 0,C 180,E1 -1881.291,E2 -1881.291} C_VEL
LIN {X 0,Y 580.222,Z 835.955,A -85,B 0,C 180,E1 -1882.167,E2 -1882.167} C_VEL
LIN {X 0,Y 580.154,Z 843.647,A -85,B 0,C 180,E1 -1883.221,E2 -1883.221} C_VEL
LIN {X 0,Y 580.139,Z 850.676,A -85,B 0,C 180,E1 -1884.438,E2 -1884.438} C_VEL
LIN {X 0,Y 580.108,Z 855.369,A -85,B 0,C 180,E1 -1885.483,E2 -1885.483} C_VEL
LIN {X 0,Y 580.123,Z 858.954,A -85,B 0,C 180,E1 -1886.527,E2 -1886.527} C_VEL
LIN {X 0,Y 580.043,Z 860.807,A -85,B 0,C 180,E1 -1887.221,E2 -1887.221} C_VEL
LIN {X 0,Y 580.038,Z 862.199,A -85,B 0,C 180,E1 -1887.916,E2 -1887.916} C_VEL
LIN {X 0,Y 580.04,Z 863.784,A -85,B 0,C 180,E1 -1889.305,E2 -1889.305} C_VEL
LIN {X 0,Y 580.037,Z 864,A -85,B 0,C 180,E1 -1889.999,E2 -1889.999} C_VEL
LIN {X 0,Y 580.047,Z 863.186,A -85,B 0,C 180,E1 -1891.388,E2 -1891.388} C_VEL
LIN {X 0,Y 580.038,Z 862.202,A -85,B 0,C 180,E1 -1892.082,E2 -1892.082} C_VEL
LIN {X 0,Y 580.043,Z 860.812,A -85,B 0,C 180,E1 -1892.777,E2 -1892.777} C_VEL
LIN {X 0,Y 580.11,Z 857.898,A -85,B 0,C 180,E1 -1893.82,E2 -1893.82} C_VEL
LIN {X 0,Y 580.054,Z 853.953,A -85,B 0,C 180,E1 -1894.864,E2 -1894.864} C_VEL
LIN {X 0,Y 580.139,Z 847.882,A -85,B 0,C 180,E1 -1896.084,E2 -1896.084} C_VEL
LIN {X 0,Y 580.184,Z 841.242,A -85,B 0,C 180,E1 -1897.132,E2 -1897.132} C_VEL
LIN {X 0,Y 580.25,Z 832.997,A -85,B 0,C 180,E1 -1898.181,E2 -1898.181} C_VEL
LIN {X 0,Y 580.307,Z 824.547,A -85,B 0,C 180,E1 -1899.058,E2 -1899.058} C_VEL
LIN {X 0,Y 580.416,Z 814.106,A -85,B 0,C 180,E1 -1899.935,E2 -1899.935} C_VEL
LIN {X 0,Y 580.512,Z 803.771,A -85,B 0,C 180,E1 -1900.638,E2 -1900.638} C_VEL
LIN {X 0,Y 580.596,Z 792.25,A -85,B 0,C 180,E1 -1901.264,E2 -1901.264} C_VEL
LIN {X 0,Y 580.673,Z 779.496,A -85,B 0,C 180,E1 -1901.784,E2 -1901.784} C_VEL
LIN {X 0,Y 580.733,Z 766.47,A -85,B 0,C 180,E1 -1902.16,E2 -1902.16} C_VEL
LIN {X 0,Y 580.846,Z 754.146,A -85,B 0,C 180,E1 -1902.379,E2 -1902.379} C_VEL
LIN {X 0,Y 580.767,Z 653.675,A -85,B 0,C 180,E1 -1903.63,E2 -1903.63} C_VEL
LIN {X 0,Y 580.441,Z 651.276,A -85,B 0,C 180,E1 -1903.678,E2 -1903.678} C_VEL
LIN {X 0,Y 580.609,Z 628.246,A -85,B 0,C 180,E1 -1906.706,E2 -1906.706} C_VEL
LIN {X 0,Y 580.826,Z 606.245,A -85,B 0,C 180,E1 -1909.641,E2 -1909.641} C_VEL
LIN {X 0,Y 581.055,Z 583.21,A -85,B 0,C 180,E1 -1912.77,E2 -1912.77} C_VEL
LIN {X 0,Y 580.987,Z 576.386,A -85,B 0,C 180,E1 -1913.716,E2 -1913.716} C_VEL
LIN {X 0,Y 580.32,Z 573.201,A -85,B 0,C 180,E1 -1914.219,E2 -1914.219} C_VEL
LIN {X 0,Y 580.278,Z 573.207,A -85,B 0,C 180,E1 -1916.622,E2 -1916.622} C_VEL
LIN {X 0,Y 580.301,Z 573.196,A -85,B 0,C 180,E1 -1919.309,E2 -1919.309} C_VEL
LIN {X 0,Y 580.297,Z 573.201,A -85,B 0,C 180,E1 -1922.199,E2 -1922.199} C_VEL
LIN {X 0,Y 580.299,Z 573.203,A -85,B 0,C 180,E1 -1924.694,E2 -1924.694} C_VEL
LIN {X 0,Y 580.296,Z 573.196,A -85,B 0,C 180,E1 -1927.267,E2 -1927.267} C_VEL
LIN {X 0,Y 580.296,Z 573.202,A -85,B 0,C 180,E1 -1930.271,E2 -1930.271} C_VEL
LIN {X 0,Y 580.274,Z 573.205,A -85,B 0,C 180,E1 -1932.705,E2 -1932.705} C_VEL
LIN {X 0,Y 580.27,Z 573.199,A -85,B 0,C 180,E1 -1935.608,E2 -1935.608} C_VEL
LIN {X 0,Y 580.31,Z 573.2,A -85,B 0,C 180,E1 -1938.234,E2 -1938.234} C_VEL
LIN {X 0,Y 580.288,Z 573.199,A -85,B 0,C 180,E1 -1940.966,E2 -1940.966} C_VEL
LIN {X 0,Y 580.291,Z 573.195,A -85,B 0,C 180,E1 -1943.598,E2 -1943.598} C_VEL
LIN {X 0,Y 580.316,Z 573.198,A -85,B 0,C 180,E1 -1946.145,E2 -1946.145} C_VEL
LIN {X 0,Y 580.285,Z 573.203,A -85,B 0,C 180,E1 -1948.615,E2 -1948.615} C_VEL
LIN {X 0,Y 580.288,Z 573.197,A -85,B 0,C 180,E1 -1951.023,E2 -1951.023} C_VEL
LIN {X 0,Y 580.323,Z 573.192,A -85,B 0,C 180,E1 -1953.658,E2 -1953.658} C_VEL
LIN {X 0,Y 580.274,Z 573.207,A -85,B 0,C 180,E1 -1956.442,E2 -1956.442} C_VEL
LIN {X 0,Y 580.269,Z 573.198,A -85,B 0,C 180,E1 -1959.437,E2 -1959.437} C_VEL
LIN {X 0,Y 580.274,Z 573.198,A -85,B 0,C 180,E1 -1961.645,E2 -1961.645} C_VEL
LIN {X 0,Y 580.273,Z 573.2,A -85,B 0,C 180,E1 -1963.825,E2 -1963.825} C_VEL
LIN {X 0,Y 580.318,Z 573.196,A -85,B 0,C 180,E1 -1965.983,E2 -1965.983} C_VEL
LIN {X 0,Y 580.296,Z 573.198,A -85,B 0,C 180,E1 -1968.827,E2 -1968.827} C_VEL
LIN {X 0,Y 580.329,Z 573.192,A -85,B 0,C 180,E1 -1971.644,E2 -1971.644} C_VEL
LIN {X 0,Y 580.316,Z 573.201,A -85,B 0,C 180,E1 -1974.44,E2 -1974.44} C_VEL
LIN {X 0,Y 580.341,Z 573.19,A -85,B 0,C 180,E1 -1977.223,E2 -1977.223} C_VEL
LIN {X 0,Y 580.344,Z 573.194,A -85,B 0,C 180,E1 -1980,E2 -1980} C_VEL
LIN {X 0,Y 580.341,Z 573.193,A -85,B 0,C 180,E1 -1982.776,E2 -1982.776} C_VEL
LIN {X 0,Y 580.324,Z 573.193,A -85,B 0,C 180,E1 -1985.56,E2 -1985.56} C_VEL
LIN {X 0,Y 580.33,Z 573.2,A -85,B 0,C 180,E1 -1988.356,E2 -1988.356} C_VEL
LIN {X 0,Y 580.325,Z 573.192,A -85,B 0,C 180,E1 -1991.208,E2 -1991.208} C_VEL
LIN {X 0,Y 580.307,Z 573.204,A -85,B 0,C 180,E1 -1994.339,E2 -1994.339} C_VEL
LIN {X 0,Y 580.319,Z 573.31,A -85,B 0,C 180,E1 -1997.474,E2 -1997.474} C_VEL
LIN {X 0,Y 580.315,Z 586.368,A -85,B 0,C 180,E1 -1999.977,E2 -1999.977} C_VEL
LIN {X 0,Y 579.712,Z 588.423,A -85,B 0,C 180,E1 -2000.336,E2 -2000.336} C_VEL
LIN {X 0,Y 577.767,Z 591.545,A -85,B 0,C 180,E1 -2000.765,E2 -2000.765} C_VEL
LIN {X 0,Y 575.59,Z 595.298,A -85,B 0,C 180,E1 -2001.107,E2 -2001.107} C_VEL
LIN {X 0,Y 574.313,Z 599.038,A -85,B 0,C 180,E1 -2001.297,E2 -2001.297} C_VEL
LIN {X 0,Y 574.064,Z 601.305,A -85,B 0,C 180,E1 -2001.349,E2 -2001.349} C_VEL
LIN {X 0,Y 573.86,Z 699.673,A -85,B 0,C 180,E1 -2002.597,E2 -2002.597} C_VEL
LIN {X 0,Y 573.784,Z 713.007,A -85,B 0,C 180,E1 -2002.909,E2 -2002.909} C_VEL
LIN {X 0,Y 573.719,Z 725.247,A -85,B 0,C 180,E1 -2003.334,E2 -2003.334} C_VEL
LIN {X 0,Y 573.584,Z 736.357,A -85,B 0,C 180,E1 -2003.85,E2 -2003.85} C_VEL
LIN {X 0,Y 573.475,Z 747.715,A -85,B 0,C 180,E1 -2004.528,E2 -2004.528} C_VEL
LIN {X 0,Y 573.368,Z 757.587,A -85,B 0,C 180,E1 -2005.261,E2 -2005.261} C_VEL
LIN {X 0,Y 573.249,Z 767.734,A -85,B 0,C 180,E1 -2006.19,E2 -2006.19} C_VEL
LIN {X 0,Y 573.164,Z 776.441,A -85,B 0,C 180,E1 -2007.178,E2 -2007.178} C_VEL
LIN {X 0,Y 573.085,Z 784.13,A -85,B 0,C 180,E1 -2008.257,E2 -2008.257} C_VEL
LIN {X 0,Y 573.071,Z 790.907,A -85,B 0,C 180,E1 -2009.459,E2 -2009.459} C_VEL
LIN {X 0,Y 573.001,Z 795.549,A -85,B 0,C 180,E1 -2010.517,E2 -2010.517} C_VEL
LIN {X 0,Y 572.95,Z 799.812,A -85,B 0,C 180,E1 -2011.833,E2 -2011.833} C_VEL
LIN {X 0,Y 572.943,Z 801.705,A -85,B 0,C 180,E1 -2012.665,E2 -2012.665} C_VEL
LIN {X 0,Y 572.958,Z 803.033,A -85,B 0,C 180,E1 -2013.503,E2 -2013.503} C_VEL
LIN {X 0,Y 572.957,Z 803.937,A -85,B 0,C 180,E1 -2014.733,E2 -2014.733} C_VEL
LIN {X 0,Y 572.923,Z 803.568,A -85,B 0,C 180,E1 -2016.073,E2 -2016.073} C_VEL
LIN {X 0,Y 572.929,Z 802.247,A -85,B 0,C 180,E1 -2017.125,E2 -2017.125} C_VEL
LIN {X 0,Y 572.973,Z 799.753,A -85,B 0,C 180,E1 -2018.28,E2 -2018.28} C_VEL
LIN {X 0,Y 572.992,Z 796.202,A -85,B 0,C 180,E1 -2019.403,E2 -2019.403} C_VEL
LIN {X 0,Y 573.035,Z 791.344,A -85,B 0,C 180,E1 -2020.543,E2 -2020.543} C_VEL
LIN {X 0,Y 573.06,Z 784.692,A -85,B 0,C 180,E1 -2021.745,E2 -2021.745} C_VEL
LIN {X 0,Y 573.139,Z 777.537,A -85,B 0,C 180,E1 -2022.772,E2 -2022.772} C_VEL
LIN {X 0,Y 573.227,Z 768.958,A -85,B 0,C 180,E1 -2023.772,E2 -2023.772} C_VEL
LIN {X 0,Y 573.335,Z 759.276,A -85,B 0,C 180,E1 -2024.688,E2 -2024.688} C_VEL
LIN {X 0,Y 573.455,Z 748.674,A -85,B 0,C 180,E1 -2025.497,E2 -2025.497} C_VEL
LIN {X 0,Y 573.576,Z 737.058,A -85,B 0,C 180,E1 -2026.203,E2 -2026.203} C_VEL
LIN {X 0,Y 573.723,Z 724.83,A -85,B 0,C 180,E1 -2026.773,E2 -2026.773} C_VEL
LIN {X 0,Y 573.794,Z 711.516,A -85,B 0,C 180,E1 -2027.225,E2 -2027.225} C_VEL
LIN {X 0,Y 573.869,Z 699.438,A -85,B 0,C 180,E1 -2027.497,E2 -2027.497} C_VEL
LIN {X 0,Y 573.955,Z 598.149,A -85,B 0,C 180,E1 -2028.783,E2 -2028.783} C_VEL
LIN {X 0,Y 573.246,Z 593.834,A -85,B 0,C 180,E1 -2028.867,E2 -2028.867} C_VEL
LIN {X 0,Y 573.394,Z 577.905,A -85,B 0,C 180,E1 -2031.94,E2 -2031.94} C_VEL
LIN {X 0,Y 573.272,Z 574.074,A -85,B 0,C 180,E1 -2032.719,E2 -2032.719} C_VEL
LIN {X 0,Y 573.272,Z 574.077,A -85,B 0,C 180,E1 -2035.673,E2 -2035.673} C_VEL
LIN {X 0,Y 573.239,Z 574.08,A -85,B 0,C 180,E1 -2038.186,E2 -2038.186} C_VEL
LIN {X 0,Y 573.262,Z 574.072,A -85,B 0,C 180,E1 -2040.635,E2 -2040.635} C_VEL
LIN {X 0,Y 573.249,Z 574.072,A -85,B 0,C 180,E1 -2043.025,E2 -2043.025} C_VEL
LIN {X 0,Y 573.273,Z 574.07,A -85,B 0,C 180,E1 -2045.367,E2 -2045.367} C_VEL
LIN {X 0,Y 573.229,Z 574.081,A -85,B 0,C 180,E1 -2048.42,E2 -2048.42} C_VEL
LIN {X 0,Y 573.278,Z 574.071,A -85,B 0,C 180,E1 -2050.729,E2 -2050.729} C_VEL
LIN {X 0,Y 573.253,Z 574.073,A -85,B 0,C 180,E1 -2053.623,E2 -2053.623} C_VEL
LIN {X 0,Y 573.275,Z 574.072,A -85,B 0,C 180,E1 -2055.808,E2 -2055.808} C_VEL
LIN {X 0,Y 573.263,Z 574.074,A -85,B 0,C 180,E1 -2058.746,E2 -2058.746} C_VEL
LIN {X 0,Y 573.286,Z 574.068,A -85,B 0,C 180,E1 -2061.541,E2 -2061.541} C_VEL
LIN {X 0,Y 573.292,Z 574.076,A -85,B 0,C 180,E1 -2064.373,E2 -2064.373} C_VEL
LIN {X 0,Y 573.314,Z 574.066,A -85,B 0,C 180,E1 -2067.893,E2 -2067.893} C_VEL
LIN {X 0,Y 573.334,Z 574.07,A -85,B 0,C 180,E1 -2070.703,E2 -2070.703} C_VEL
LIN {X 0,Y 573.312,Z 574.071,A -85,B 0,C 180,E1 -2072.811,E2 -2072.811} C_VEL
LIN {X 0,Y 573.291,Z 574.067,A -85,B 0,C 180,E1 -2075.629,E2 -2075.629} C_VEL
LIN {X 0,Y 573.293,Z 574.073,A -85,B 0,C 180,E1 -2078.46,E2 -2078.46} C_VEL
LIN {X 0,Y 573.275,Z 574.071,A -85,B 0,C 180,E1 -2081.313,E2 -2081.313} C_VEL
LIN {X 0,Y 573.277,Z 574.07,A -85,B 0,C 180,E1 -2084.194,E2 -2084.194} C_VEL
LIN {X 0,Y 573.262,Z 574.077,A -85,B 0,C 180,E1 -2087.112,E2 -2087.112} C_VEL
LIN {X 0,Y 573.247,Z 574.073,A -85,B 0,C 180,E1 -2090.077,E2 -2090.077} C_VEL
LIN {X 0,Y 573.239,Z 574.075,A -85,B 0,C 180,E1 -2092.338,E2 -2092.338} C_VEL
LIN {X 0,Y 573.258,Z 574.075,A -85,B 0,C 180,E1 -2095.411,E2 -2095.411} C_VEL
LIN {X 0,Y 573.256,Z 574.071,A -85,B 0,C 180,E1 -2098.03,E2 -2098.03} C_VEL
LIN {X 0,Y 573.249,Z 574.072,A -85,B 0,C 180,E1 -2100.177,E2 -2100.177} C_VEL
LIN {X 0,Y 573.258,Z 574.074,A -85,B 0,C 180,E1 -2102.645,E2 -2102.645} C_VEL
LIN {X 0,Y 573.244,Z 574.084,A -85,B 0,C 180,E1 -2105.186,E2 -2105.186} C_VEL
LIN {X 0,Y 573.239,Z 574.075,A -85,B 0,C 180,E1 -2107.808,E2 -2107.808} C_VEL
LIN {X 0,Y 573.248,Z 574.073,A -85,B 0,C 180,E1 -2110.525,E2 -2110.525} C_VEL
LIN {X 0,Y 573.241,Z 574.084,A -85,B 0,C 180,E1 -2113.36,E2 -2113.36} C_VEL
LIN {X 0,Y 573.249,Z 574.072,A -85,B 0,C 180,E1 -2116.331,E2 -2116.331} C_VEL
LIN {X 0,Y 573.244,Z 574.073,A -85,B 0,C 180,E1 -2118.544,E2 -2118.544} C_VEL
LIN {X 0,Y 573.248,Z 574.08,A -85,B 0,C 180,E1 -2121.299,E2 -2121.299} C_VEL
LIN {X 0,Y 573.217,Z 574.079,A -85,B 0,C 180,E1 -2124.019,E2 -2124.019} C_VEL
LIN {X 0,Y 573.274,Z 574.069,A -85,B 0,C 180,E1 -2126.518,E2 -2126.518} C_VEL
LIN {X 0,Y 573.233,Z 574.077,A -85,B 0,C 180,E1 -2129.118,E2 -2129.118} C_VEL
LIN {X 0,Y 573.243,Z 574.079,A -85,B 0,C 180,E1 -2131.436,E2 -2131.436} C_VEL
LIN {X 0,Y 573.268,Z 574.079,A -85,B 0,C 180,E1 -2133.81,E2 -2133.81} C_VEL
LIN {X 0,Y 573.232,Z 574.079,A -85,B 0,C 180,E1 -2136.135,E2 -2136.135} C_VEL
LIN {X 0,Y 573.256,Z 574.073,A -85,B 0,C 180,E1 -2139.174,E2 -2139.174} C_VEL
LIN {X 0,Y 573.224,Z 574.079,A -85,B 0,C 180,E1 -2141.411,E2 -2141.411} C_VEL
LIN {X 0,Y 573.254,Z 574.077,A -85,B 0,C 180,E1 -2143.622,E2 -2143.622} C_VEL
LIN {X 0,Y 573.278,Z 574.077,A -85,B 0,C 180,E1 -2145.807,E2 -2145.807} C_VEL
LIN {X 0,Y 573.268,Z 574.07,A -85,B 0,C 180,E1 -2148.745,E2 -2148.745} C_VEL
LIN {X 0,Y 573.289,Z 574.07,A -85,B 0,C 180,E1 -2151.541,E2 -2151.541} C_VEL
LIN {X 0,Y 573.292,Z 574.072,A -85,B 0,C 180,E1 -2154.372,E2 -2154.372} C_VEL
LIN {X 0,Y 573.315,Z 574.07,A -85,B 0,C 180,E1 -2157.893,E2 -2157.893} C_VEL
LIN {X 0,Y 573.336,Z 574.064,A -85,B 0,C 180,E1 -2160.702,E2 -2160.702} C_VEL
LIN {X 0,Y 573.235,Z 574.075,A -85,B 0,C 180,E1 -2163.515,E2 -2163.515} C_VEL
LIN {X 0,Y 573.289,Z 574.068,A -85,B 0,C 180,E1 -2165.628,E2 -2165.628} C_VEL
LIN {X 0,Y 573.289,Z 574.076,A -85,B 0,C 180,E1 -2168.46,E2 -2168.46} C_VEL
LIN {X 0,Y 573.278,Z 574.069,A -85,B 0,C 180,E1 -2171.312,E2 -2171.312} C_VEL
LIN {X 0,Y 573.287,Z 574.078,A -85,B 0,C 180,E1 -2174.424,E2 -2174.424} C_VEL
LIN {X 0,Y 573.264,Z 574.072,A -85,B 0,C 180,E1 -2177.112,E2 -2177.112} C_VEL
LIN {X 0,Y 573.248,Z 574.075,A -85,B 0,C 180,E1 -2180.077,E2 -2180.077} C_VEL
LIN {X 0,Y 573.239,Z 574.079,A -85,B 0,C 180,E1 -2182.338,E2 -2182.338} C_VEL
LIN {X 0,Y 573.254,Z 574.072,A -85,B 0,C 180,E1 -2185.41,E2 -2185.41} C_VEL
LIN {X 0,Y 573.252,Z 574.073,A -85,B 0,C 180,E1 -2188.028,E2 -2188.028} C_VEL
LIN {X 0,Y 573.251,Z 574.074,A -85,B 0,C 180,E1 -2190.176,E2 -2190.176} C_VEL
LIN {X 0,Y 573.258,Z 574.079,A -85,B 0,C 180,E1 -2192.645,E2 -2192.645} C_VEL
LIN {X 0,Y 573.214,Z 574.081,A -85,B 0,C 180,E1 -2195.188,E2 -2195.188} C_VEL
LIN {X 0,Y 573.241,Z 574.073,A -85,B 0,C 180,E1 -2197.807,E2 -2197.807} C_VEL
LIN {X 0,Y 573.25,Z 574.076,A -85,B 0,C 180,E1 -2200.525,E2 -2200.525} C_VEL
LIN {X 0,Y 573.246,Z 574.077,A -85,B 0,C 180,E1 -2203.359,E2 -2203.359} C_VEL
LIN {X 0,Y 573.244,Z 574.074,A -85,B 0,C 180,E1 -2206.331,E2 -2206.331} C_VEL
LIN {X 0,Y 573.234,Z 574.076,A -85,B 0,C 180,E1 -2208.543,E2 -2208.543} C_VEL
LIN {X 0,Y 573.25,Z 574.08,A -85,B 0,C 180,E1 -2211.298,E2 -2211.298} C_VEL
LIN {X 0,Y 573.22,Z 574.076,A -85,B 0,C 180,E1 -2214.018,E2 -2214.018} C_VEL
LIN {X 0,Y 573.292,Z 574.068,A -85,B 0,C 180,E1 -2216.519,E2 -2216.519} C_VEL
LIN {X 0,Y 573.229,Z 574.083,A -85,B 0,C 180,E1 -2219.118,E2 -2219.118} C_VEL
LIN {X 0,Y 573.243,Z 574.083,A -85,B 0,C 180,E1 -2221.435,E2 -2221.435} C_VEL
LIN {X 0,Y 573.265,Z 574.076,A -85,B 0,C 180,E1 -2223.81,E2 -2223.81} C_VEL
LIN {X 0,Y 573.302,Z 574.156,A -85,B 0,C 180,E1 -2225.632,E2 -2225.632} C_VEL
LIN {X 0,Y 574.205,Z 579.997,A -85,B 0,C 180,E1 -2226.494,E2 -2226.494} C_VEL
LIN {X 0,Y 573.954,Z 599.575,A -85,B 0,C 180,E1 -2229.2,E2 -2229.2} C_VEL
LIN {X 0,Y 573.706,Z 621.41,A -85,B 0,C 180,E1 -2232.166,E2 -2232.166} C_VEL
LIN {X 0,Y 573.493,Z 643.246,A -85,B 0,C 180,E1 -2235.086,E2 -2235.086} C_VEL
LIN {X 0,Y 573.439,Z 651.349,A -85,B 0,C 180,E1 -2236.161,E2 -2236.161} C_VEL
LIN {X 0,Y 574.084,Z 657.453,A -85,B 0,C 180,E1 -2236.256,E2 -2236.256} C_VEL
LIN {X 0,Y 573.897,Z 759.91,A -85,B 0,C 180,E1 -2237.557,E2 -2237.557} C_VEL
LIN {X 0,Y 573.801,Z 772.434,A -85,B 0,C 180,E1 -2237.847,E2 -2237.847} C_VEL
LIN {X 0,Y 573.706,Z 785.355,A -85,B 0,C 180,E1 -2238.293,E2 -2238.293} C_VEL
LIN {X 0,Y 573.58,Z 797.708,A -85,B 0,C 180,E1 -2238.878,E2 -2238.878} C_VEL
LIN {X 0,Y 573.441,Z 809.193,A -85,B 0,C 180,E1 -2239.584,E2 -2239.584} C_VEL
LIN {X 0,Y 573.327,Z 819.591,A -85,B 0,C 180,E1 -2240.385,E2 -2240.385} C_VEL
LIN {X 0,Y 573.239,Z 828.105,A -85,B 0,C 180,E1 -2241.184,E2 -2241.184} C_VEL
LIN {X 0,Y 573.161,Z 835.955,A -85,B 0,C 180,E1 -2242.07,E2 -2242.07} C_VEL
LIN {X 0,Y 573.073,Z 843.951,A -85,B 0,C 180,E1 -2243.185,E2 -2243.185} C_VEL
LIN {X 0,Y 573.07,Z 850.676,A -85,B 0,C 180,E1 -2244.369,E2 -2244.369} C_VEL
LIN {X 0,Y 573.029,Z 855.369,A -85,B 0,C 180,E1 -2245.427,E2 -2245.427} C_VEL
LIN {X 0,Y 573.023,Z 858.955,A -85,B 0,C 180,E1 -2246.483,E2 -2246.483} C_VEL
LIN {X 0,Y 572.959,Z 860.807,A -85,B 0,C 180,E1 -2247.187,E2 -2247.187} C_VEL
LIN {X 0,Y 572.937,Z 862.198,A -85,B 0,C 180,E1 -2247.89,E2 -2247.89} C_VEL
LIN {X 0,Y 572.941,Z 863.784,A -85,B 0,C 180,E1 -2249.296,E2 -2249.296} C_VEL
LIN {X 0,Y 572.938,Z 864,A -85,B 0,C 180,E1 -2249.999,E2 -2249.999} C_VEL
LIN {X 0,Y 572.946,Z 863.187,A -85,B 0,C 180,E1 -2251.405,E2 -2251.405} C_VEL
LIN {X 0,Y 572.937,Z 862.201,A -85,B 0,C 180,E1 -2252.108,E2 -2252.108} C_VEL
LIN {X 0,Y 572.959,Z 860.812,A -85,B 0,C 180,E1 -2252.812,E2 -2252.812} C_VEL
LIN {X 0,Y 573.014,Z 857.898,A -85,B 0,C 180,E1 -2253.867,E2 -2253.867} C_VEL
LIN {X 0,Y 572.963,Z 853.952,A -85,B 0,C 180,E1 -2254.925,E2 -2254.925} C_VEL
LIN {X 0,Y 573.064,Z 847.882,A -85,B 0,C 180,E1 -2256.159,E2 -2256.159} C_VEL
LIN {X 0,Y 573.119,Z 841.243,A -85,B 0,C 180,E1 -2257.22,E2 -2257.22} C_VEL
LIN {X 0,Y 573.2,Z 832.997,A -85,B 0,C 180,E1 -2258.282,E2 -2258.282} C_VEL
LIN {X 0,Y 573.286,Z 824.547,A -85,B 0,C 180,E1 -2259.169,E2 -2259.169} C_VEL
LIN {X 0,Y 573.422,Z 814.108,A -85,B 0,C 180,E1 -2260.058,E2 -2260.058} C_VEL
LIN {X 0,Y 573.548,Z 802.367,A -85,B 0,C 180,E1 -2260.857,E2 -2260.857} C_VEL
LIN {X 0,Y 573.651,Z 791.299,A -85,B 0,C 180,E1 -2261.446,E2 -2261.446} C_VEL
LIN {X 0,Y 573.771,Z 778.198,A -85,B 0,C 180,E1 -2261.973,E2 -2261.973} C_VEL
LIN {X 0,Y 573.805,Z 765.555,A -85,B 0,C 180,E1 -2262.331,E2 -2262.331} C_VEL
LIN {X 0,Y 573.901,Z 752.378,A -85,B 0,C 180,E1 -2262.554,E2 -2262.554} C_VEL
LIN {X 0,Y 573.95,Z 654.896,A -85,B 0,C 180,E1 -2263.78,E2 -2263.78} C_VEL
LIN {X 0,Y 573.445,Z 651.276,A -85,B 0,C 180,E1 -2263.848,E2 -2263.848} C_VEL
LIN {X 0,Y 573.635,Z 628.252,A -85,B 0,C 180,E1 -2266.915,E2 -2266.915} C_VEL
LIN {X 0,Y 573.884,Z 607.774,A -85,B 0,C 180,E1 -2269.68,E2 -2269.68} C_VEL
LIN {X 0,Y 574.159,Z 584.574,A -85,B 0,C 180,E1 -2272.869,E2 -2272.869} C_VEL
LIN {X 0,Y 574.052,Z 577.751,A -85,B 0,C 180,E1 -2273.828,E2 -2273.828} C_VEL
LIN {X 0,Y 573.286,Z 574.078,A -85,B 0,C 180,E1 -2274.391,E2 -2274.391} C_VEL
LIN {X 0,Y 573.251,Z 574.078,A -85,B 0,C 180,E1 -2276.975,E2 -2276.975} C_VEL
LIN {X 0,Y 573.246,Z 574.074,A -85,B 0,C 180,E1 -2279.487,E2 -2279.487} C_VEL
LIN {X 0,Y 573.253,Z 574.082,A -85,B 0,C 180,E1 -2282.644,E2 -2282.644} C_VEL
LIN {X 0,Y 573.266,Z 574.073,A -85,B 0,C 180,E1 -2285.183,E2 -2285.183} C_VEL
LIN {X 0,Y 573.233,Z 574.076,A -85,B 0,C 180,E1 -2287.807,E2 -2287.807} C_VEL
LIN {X 0,Y 573.266,Z 574.081,A -85,B 0,C 180,E1 -2290.527,E2 -2290.527} C_VEL
LIN {X 0,Y 573.24,Z 574.075,A -85,B 0,C 180,E1 -2293.668,E2 -2293.668} C_VEL
LIN {X 0,Y 573.243,Z 574.082,A -85,B 0,C 180,E1 -2296.641,E2 -2296.641} C_VEL
LIN {X 0,Y 573.269,Z 574.07,A -85,B 0,C 180,E1 -2299.477,E2 -2299.477} C_VEL
LIN {X 0,Y 573.234,Z 574.08,A -85,B 0,C 180,E1 -2302.192,E2 -2302.192} C_VEL
LIN {X 0,Y 573.263,Z 574.075,A -85,B 0,C 180,E1 -2304.816,E2 -2304.816} C_VEL
